// TIA Portal project "Plantilla_eProC" (V15.1)

(* hardware
DEVICE "S7-1200 station_1"  S7-1200 Station
   slot 0: "Rack_0"  S7-1200 Rack  Rack  V1.0
   slot 1: "PLC_1"  CPU 1214C DC/DC/DC  6ES7 214-1AG40-0XB0  V4.3
*)

// ===== PLC "PLC_1"  CPU 1214C DC/DC/DC =====

VAR_GLOBAL   // PLC tag table "Tabla de variables estándar"
   "System_Byte" AT %MB1 : Byte;
   "FirstScan" AT %M1.0 : Bool;
   "DiagStatusUpdate" AT %M1.1 : Bool;
   "AlwaysTRUE" AT %M1.2 : Bool;
   "AlwaysFALSE" AT %M1.3 : Bool;
   "Clock_Byte" AT %MB0 : Byte;
   "Clock_10Hz" AT %M0.0 : Bool;
   "Clock_5Hz" AT %M0.1 : Bool;
   "Clock_2.5Hz" AT %M0.2 : Bool;
   "Clock_2Hz" AT %M0.3 : Bool;
   "Clock_1.25Hz" AT %M0.4 : Bool;
   "Clock_1Hz" AT %M0.5 : Bool;
   "Clock_0.625Hz" AT %M0.6 : Bool;
   "Clock_0.5Hz" AT %M0.7 : Bool;
   "Marca_Manual" AT %M2.0 : Bool;
   "Marca_Automatico" AT %M2.1 : Bool;
   "Tim_Extrac_Rdy" AT %M3.0 : Bool;
   "Tim_Induc_Rdy" AT %M3.1 : Bool;
   "B_TimAperturaLados" AT %M4.0 : Bool;
END_VAR

VAR_GLOBAL   // PLC tag table "Entradas_PLC"
   "iPul_ParEmergencia" AT %I0.0 : Bool;
   "iSel_CicloManual" AT %I0.1 : Bool;
   "iSel_CicloAuto" AT %I0.2 : Bool;
   "iSel_AvanzCamaRolos1" AT %I0.3 : Bool;
   "iSel_RetroCamaRolos1" AT %I0.4 : Bool;
   "iSel_AvanzCamaRolos2" AT %I0.5 : Bool;
   "iSel_RetroCamaRolos2" AT %I0.6 : Bool;
   "iReserva1" AT %I0.7 : Bool;
   "iProt_TermicaRolos" AT %I1.0 : Bool;
   "iStart_CicloDesdeSoldad" AT %I1.1 : Bool;
   "iSns_PresAire" AT %I1.2 : Bool;
   "iReserva2" AT %I1.3 : Bool;
   "iReserva3" AT %I1.4 : Bool;
   "iReserva4" AT %I1.5 : Bool;
   "iSns_ElevArriba" AT %I2.0 : Bool;
   "iSns_ElevAbajo" AT %I2.1 : Bool;
   "iSns_ElevNormal" AT %I2.2 : Bool;
   "iSns_ElevRotado" AT %I2.3 : Bool;
   "iSns_PreseProduc" AT %I2.4 : Bool;
   "iSns_CR1LadoTableroArri" AT %I2.5 : Bool;
   "iSns_CR1LadoTableroAbaj" AT %I2.6 : Bool;
   "iSns_RegAlturaPaq" AT %I2.7 : Bool;
   "iSns_CR1LadoOpuesArri" AT %I3.0 : Bool;
   "iSns_CR1LadoOpuesAbaj" AT %I3.1 : Bool;
   "iSns_PreseProducSalida1" AT %I3.2 : Bool;
   "iSns_PreseProducSalida2" AT %I3.3 : Bool;
   "iPul_StartCiclo" AT %I3.4 : Bool;
   "iSel_HabRuedExtrac" AT %I3.5 : Bool;
   "iPul_MarchRuedExtrac" AT %I3.6 : Bool;
   "iReserva5" AT %I3.7 : Bool;
   "iSel_HabRuedIntroduc" AT %I4.0 : Bool;
   "iPul_MarchRuedIntroduc" AT %I4.1 : Bool;
END_VAR

VAR_GLOBAL   // PLC tag table "Salidas_PLC"
   "qCR1_LTArri" AT %Q0.0 : Bool;
   "qCR1_LTAbaj" AT %Q0.1 : Bool;
   "qCR1_LOArri" AT %Q0.2 : Bool;
   "qCR1_LOAbaj" AT %Q0.3 : Bool;
   "qCR1_Avance" AT %Q0.4 : Bool;
   "qCR1_Retroceso" AT %Q0.5 : Bool;
   "qCR2_Avance" AT %Q0.6 : Bool;
   "qCR2_Retroceso" AT %Q0.7 : Bool;
   "qHab_Comandos" AT %Q1.0 : Bool;
   "qRdy_VoltRdyaSold" AT %Q1.1 : Bool;
   "qBrk_Volt" AT %Q2.0 : Bool;
   "qBrk_Elev" AT %Q2.1 : Bool;
   "qCls_RodExtrac" AT %Q2.2 : Bool;
   "qCls_RodInduc" AT %Q2.3 : Bool;
   "qCls_Ganchos" AT %Q2.4 : Bool;
   "qOpn_Lados" AT %Q2.5 : Bool;
   "qAcc_Compact" AT %Q2.6 : Bool;
   "qCls_SoportRed" AT %Q2.7 : Bool;
END_VAR

DATA_BLOCK "DB_SUB_0_GENERAL"   // DB100
{ S7_Optimized_Access := 'TRUE' }
VERSION : 0.1
// stored: InstanceOfName FB_SUB_0_GENERAL
"FB_SUB_0_GENERAL"
BEGIN
END_DATA_BLOCK

DATA_BLOCK "DB_SUB_1_ELEVADOR"   // DB101
{ S7_Optimized_Access := 'TRUE' }
VERSION : 0.1
// stored: InstanceOfName FB_SUB_1_ELEVADOR
"FB_SUB_1_ELEVADOR"
BEGIN
END_DATA_BLOCK

DATA_BLOCK "DB_SUB_1_CAMAS_ROLOS"   // DB102
{ S7_Optimized_Access := 'TRUE' }
VERSION : 0.1
// stored: InstanceOfName FB_SUB_1_CAMAS_ROLOS
"FB_SUB_1_CAMAS_ROLOS"
BEGIN
END_DATA_BLOCK

DATA_BLOCK "DB_SUB_1_MAQUINA_ESTADOS_3"   // DB103
{ S7_Optimized_Access := 'TRUE' }
VERSION : 0.1
// stored: InstanceOfName FB_SUB_1_MAQUINA_ESTADOS_3
"FB_SUB_1_MAQUINA_ESTADOS_3"
BEGIN
END_DATA_BLOCK

DATA_BLOCK "DB_SUB_1_MAQUINA_ESTADOS_4"   // DB104
{ S7_Optimized_Access := 'TRUE' }
VERSION : 0.1
// stored: InstanceOfName FB_SUB_1_MAQUINA_ESTADOS_4
"FB_SUB_1_MAQUINA_ESTADOS_4"
BEGIN
END_DATA_BLOCK

// folder: AJUSTE_PEM

DATA_BLOCK "DB_SUB_0_PEM_GENERAL"   // DB400
{ S7_Optimized_Access := 'TRUE' }
VERSION : 0.1
BEGIN
END_DATA_BLOCK

DATA_BLOCK "DB_SUB_1_PEM_MAQ_ESTADO_1"   // DB401
{ S7_Optimized_Access := 'TRUE' }
VERSION : 0.1
BEGIN
END_DATA_BLOCK

DATA_BLOCK "DB_SUB_1_PEM_MAQ_ESTADO_2"   // DB402
{ S7_Optimized_Access := 'TRUE' }
VERSION : 0.1
BEGIN
END_DATA_BLOCK

DATA_BLOCK "DB_SUB_1_PEM_MAQ_ESTADO_3"   // DB403
{ S7_Optimized_Access := 'TRUE' }
VERSION : 0.1
BEGIN
END_DATA_BLOCK

DATA_BLOCK "DB_SUB_1_PEM_MAQ_ESTADO_4"   // DB404
{ S7_Optimized_Access := 'TRUE' }
VERSION : 0.1
BEGIN
END_DATA_BLOCK

// folder: COMANDOS

DATA_BLOCK "DB_SUB_0_COM_GENERAL"   // DB600
{ S7_Optimized_Access := 'TRUE' }
VERSION : 0.1
BEGIN
END_DATA_BLOCK

DATA_BLOCK "DB_SUB_1_COM_MAQ_ESTADO_1"   // DB601
{ S7_Optimized_Access := 'TRUE' }
VERSION : 0.1
BEGIN
END_DATA_BLOCK

DATA_BLOCK "DB_SUB_1_COM_MAQ_ESTADO_2"   // DB602
{ S7_Optimized_Access := 'TRUE' }
VERSION : 0.1
BEGIN
END_DATA_BLOCK

DATA_BLOCK "DB_SUB_1_COM_MAQ_ESTADO_3"   // DB603
{ S7_Optimized_Access := 'TRUE' }
VERSION : 0.1
BEGIN
END_DATA_BLOCK

DATA_BLOCK "DB_SUB_1_COM_MAQ_ESTADO_4"   // DB604
{ S7_Optimized_Access := 'TRUE' }
VERSION : 0.1
BEGIN
END_DATA_BLOCK

// folder: ENCLAVAMIENTOS

DATA_BLOCK "DB_SUB_0_ENC_GENERAL"   // DB700
{ S7_Optimized_Access := 'TRUE' }
VERSION : 0.1
BEGIN
END_DATA_BLOCK

DATA_BLOCK "DB_SUB_1_ENC_MAQ_ESTADOS_1"   // DB701
{ S7_Optimized_Access := 'TRUE' }
VERSION : 0.1
BEGIN
END_DATA_BLOCK

DATA_BLOCK "DB_SUB_1_ENC_MAQ_ESTADOS_2"   // DB702
{ S7_Optimized_Access := 'TRUE' }
VERSION : 0.1
BEGIN
END_DATA_BLOCK

DATA_BLOCK "DB_SUB_1_ENC_MAQ_ESTADOS_3"   // DB703
{ S7_Optimized_Access := 'TRUE' }
VERSION : 0.1
BEGIN
END_DATA_BLOCK

DATA_BLOCK "DB_SUB_1_ENC_MAQ_ESTADOS_4"   // DB704
{ S7_Optimized_Access := 'TRUE' }
VERSION : 0.1
BEGIN
END_DATA_BLOCK

// folder: ESTANDAR

DATA_BLOCK "Datos PLC"   // DB4
{ S7_Optimized_Access := 'TRUE' }
VERSION : 0.1
   VAR
      FH_Setpoint : DTL;   // Fecha y Hora del PLC
      FH : DTL;   // Fecha y Hora del PLC
      COM_Ajuste_FH : Bool;
   END_VAR
BEGIN
END_DATA_BLOCK

// folder: INCIDENTES

DATA_BLOCK "DB_SUB_0_GENERAL_ALARM"   // DB1100
{ S7_Optimized_Access := 'TRUE' }
VERSION : 0.1
// stored: InstanceOfName FB_SUB_0_GENERAL_ALARM
"FB_SUB_0_GENERAL_ALARM"
BEGIN
END_DATA_BLOCK

DATA_BLOCK "DB_SUB_1_MAQ_ESTADO_1_ALARM"   // DB1101
{ S7_Optimized_Access := 'TRUE' }
VERSION : 0.1
// stored: InstanceOfName FB_SUB_1_MAQ_ESTADO_1_ALARM
"FB_SUB_1_MAQ_ESTADO_1_ALARM"
BEGIN
END_DATA_BLOCK

DATA_BLOCK "DB_SUB_1_MAQ_ESTADO_2_ALARM"   // DB1102
{ S7_Optimized_Access := 'TRUE' }
VERSION : 0.1
// stored: InstanceOfName FB_SUB_1_MAQ_ESTADO_2_ALARM
"FB_SUB_1_MAQ_ESTADO_2_ALARM"
BEGIN
END_DATA_BLOCK

DATA_BLOCK "DB_SUB_1_MAQ_ESTADO_3_ALARM"   // DB1103
{ S7_Optimized_Access := 'TRUE' }
VERSION : 0.1
// stored: InstanceOfName FB_SUB_1_MAQ_ESTADO_3_ALARM
"FB_SUB_1_MAQ_ESTADO_3_ALARM"
BEGIN
END_DATA_BLOCK

DATA_BLOCK "DB_SUB_1_MAQ_ESTADO_4_ALARM"   // DB1104
{ S7_Optimized_Access := 'TRUE' }
VERSION : 0.1
// stored: InstanceOfName FB_SUB_1_MAQ_ESTADO_4_ALARM
"FB_SUB_1_MAQ_ESTADO_4_ALARM"
BEGIN
END_DATA_BLOCK

// folder: MECANICA

DATA_BLOCK "DB_SUB_0_MEC_GENERAL"   // DB300
{ S7_Optimized_Access := 'TRUE' }
VERSION : 0.1
BEGIN
END_DATA_BLOCK

DATA_BLOCK "DB_SUB_1_MEC_MAQ_ESTADO_1"   // DB301
{ S7_Optimized_Access := 'TRUE' }
VERSION : 0.1
BEGIN
END_DATA_BLOCK

DATA_BLOCK "DB_SUB_1_MEC_MAQ_ESTADO_2"   // DB302
{ S7_Optimized_Access := 'TRUE' }
VERSION : 0.1
BEGIN
END_DATA_BLOCK

DATA_BLOCK "DB_SUB_1_MEC_MAQ_ESTADO_3"   // DB303
{ S7_Optimized_Access := 'TRUE' }
VERSION : 0.1
BEGIN
END_DATA_BLOCK

DATA_BLOCK "DB_SUB_1_MEC_MAQ_ESTADO_4"   // DB304
{ S7_Optimized_Access := 'TRUE' }
VERSION : 0.1
BEGIN
END_DATA_BLOCK

// folder: System blocks/Program resources

DATA_BLOCK "IEC_Timer_0_DB"   // DB1
{ S7_Optimized_Access := 'TRUE' }
AUTHOR : Simatic
FAMILY : IEC
NAME : IEC_TMR
VERSION : 1.0
// stored: InstanceOfName IEC_TIMER
"IEC_TIMER"
BEGIN
END_DATA_BLOCK

DATA_BLOCK "IEC_Timer_1_DB"   // DB2
{ S7_Optimized_Access := 'TRUE' }
AUTHOR : Simatic
FAMILY : IEC
NAME : IEC_TMR
VERSION : 1.0
// stored: InstanceOfName IEC_TIMER
"IEC_TIMER"
BEGIN
END_DATA_BLOCK

DATA_BLOCK "IEC_Timer_2_DB"   // DB3
{ S7_Optimized_Access := 'TRUE' }
AUTHOR : Simatic
FAMILY : IEC
NAME : IEC_TMR
VERSION : 1.0
// stored: InstanceOfName IEC_TIMER
"IEC_TIMER"
BEGIN
END_DATA_BLOCK

DATA_BLOCK "IEC_Timer_3_DB"   // DB5
{ S7_Optimized_Access := 'TRUE' }
AUTHOR : Simatic
FAMILY : IEC
NAME : IEC_TMR
VERSION : 1.0
// stored: InstanceOfName IEC_TIMER
"IEC_TIMER"
BEGIN
END_DATA_BLOCK

DATA_BLOCK "IEC_Timer_5_DB"   // DB6
{ S7_Optimized_Access := 'TRUE' }
AUTHOR : Simatic
FAMILY : IEC
NAME : IEC_TMR
VERSION : 1.0
// stored: InstanceOfName IEC_TIMER
"IEC_TIMER"
BEGIN
END_DATA_BLOCK

DATA_BLOCK "IEC_Timer_6_DB"   // DB7
{ S7_Optimized_Access := 'TRUE' }
AUTHOR : Simatic
FAMILY : IEC
NAME : IEC_TMR
VERSION : 1.0
// stored: InstanceOfName IEC_TIMER
"IEC_TIMER"
BEGIN
END_DATA_BLOCK

DATA_BLOCK "IEC_Timer_7_DB"   // DB8
{ S7_Optimized_Access := 'TRUE' }
AUTHOR : Simatic
FAMILY : IEC
NAME : IEC_TMR
VERSION : 1.0
// stored: InstanceOfName IEC_TIMER
"IEC_TIMER"
BEGIN
END_DATA_BLOCK

// folder: VISUALIZACION

DATA_BLOCK "DB_SUB_0_VIS_GENERAL"   // DB800
{ S7_Optimized_Access := 'TRUE' }
VERSION : 0.1
BEGIN
END_DATA_BLOCK

DATA_BLOCK "DB_SUB_1_VIS_MAQ_ESTADO_1"   // DB801
{ S7_Optimized_Access := 'TRUE' }
VERSION : 0.1
BEGIN
END_DATA_BLOCK

DATA_BLOCK "DB_SUB_1_VIS_MAQ_ESTADO_2"   // DB802
{ S7_Optimized_Access := 'TRUE' }
VERSION : 0.1
BEGIN
END_DATA_BLOCK

DATA_BLOCK "DB_SUB_1_VIS_MAQ_ESTADO_3"   // DB803
{ S7_Optimized_Access := 'TRUE' }
VERSION : 0.1
BEGIN
END_DATA_BLOCK

DATA_BLOCK "DB_SUB_1_VIS_MAQ_ESTADO_4"   // DB804
{ S7_Optimized_Access := 'TRUE' }
VERSION : 0.1
BEGIN
END_DATA_BLOCK

// folder: (top level)

FUNCTION_BLOCK "FB_SUB_0_GENERAL"   // FB100, LAD
{ S7_Optimized_Access := 'TRUE' }
VERSION : 0.1
BEGIN

REGION Network 1: Instanciado Bloque "FB_SUB_1_MAQUINA_ESTADOS_1"
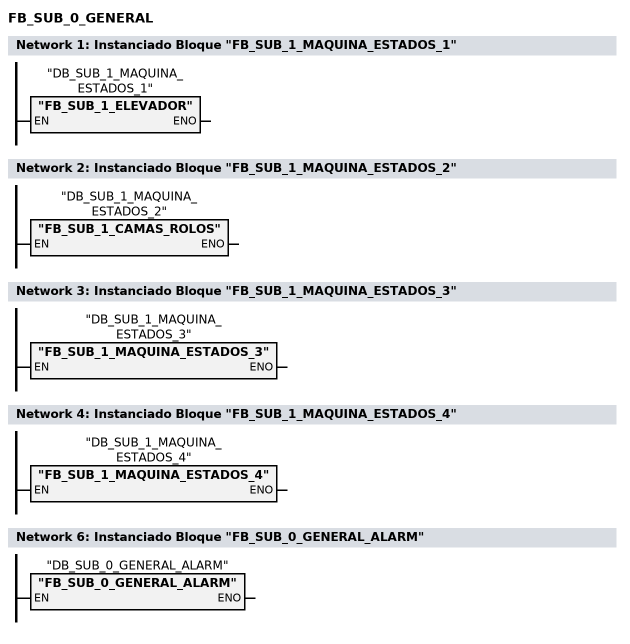
   RUNG wire#powerrail
      "DB_SUB_1_MAQUINA_ESTADOS_1"()
   END_RUNG
   // the same network as SCL:
   "DB_SUB_1_MAQUINA_ESTADOS_1"();   // "FB_SUB_1_ELEVADOR"
END_REGION

REGION Network 2: Instanciado Bloque "FB_SUB_1_MAQUINA_ESTADOS_2"
   RUNG wire#powerrail
      "DB_SUB_1_MAQUINA_ESTADOS_2"()
   END_RUNG
   // the same network as SCL:
   "DB_SUB_1_MAQUINA_ESTADOS_2"();   // "FB_SUB_1_CAMAS_ROLOS"
END_REGION

REGION Network 3: Instanciado Bloque "FB_SUB_1_MAQUINA_ESTADOS_3"
   RUNG wire#powerrail
      "DB_SUB_1_MAQUINA_ESTADOS_3"()
   END_RUNG
   // the same network as SCL:
   "DB_SUB_1_MAQUINA_ESTADOS_3"();   // "FB_SUB_1_MAQUINA_ESTADOS_3"
END_REGION

REGION Network 4: Instanciado Bloque "FB_SUB_1_MAQUINA_ESTADOS_4"
   RUNG wire#powerrail
      "DB_SUB_1_MAQUINA_ESTADOS_4"()
   END_RUNG
   // the same network as SCL:
   "DB_SUB_1_MAQUINA_ESTADOS_4"();   // "FB_SUB_1_MAQUINA_ESTADOS_4"
END_REGION

REGION Network 5: ---------------------------------------------------------------------------------------------------------
END_REGION

REGION Network 6: Instanciado Bloque "FB_SUB_0_GENERAL_ALARM"
   RUNG wire#powerrail
      "DB_SUB_0_GENERAL_ALARM"()
   END_RUNG
   // the same network as SCL:
   "DB_SUB_0_GENERAL_ALARM"();   // "FB_SUB_0_GENERAL_ALARM"
END_REGION
END_FUNCTION_BLOCK

FUNCTION_BLOCK "FB_SUB_1_ELEVADOR"   // FB101, LAD
{ S7_Optimized_Access := 'TRUE' }
VERSION : 0.1
   VAR
      Estados : Array[0..32] of Bool;
      Concatenadoras : Array[0..32] of Bool;
      Prioritarias : Array[0..32] of Bool;
   END_VAR
BEGIN

REGION Network 1: --------------------------------------INSTANCIADO DE SUBSISTEMAS ---------------------------------------------------------
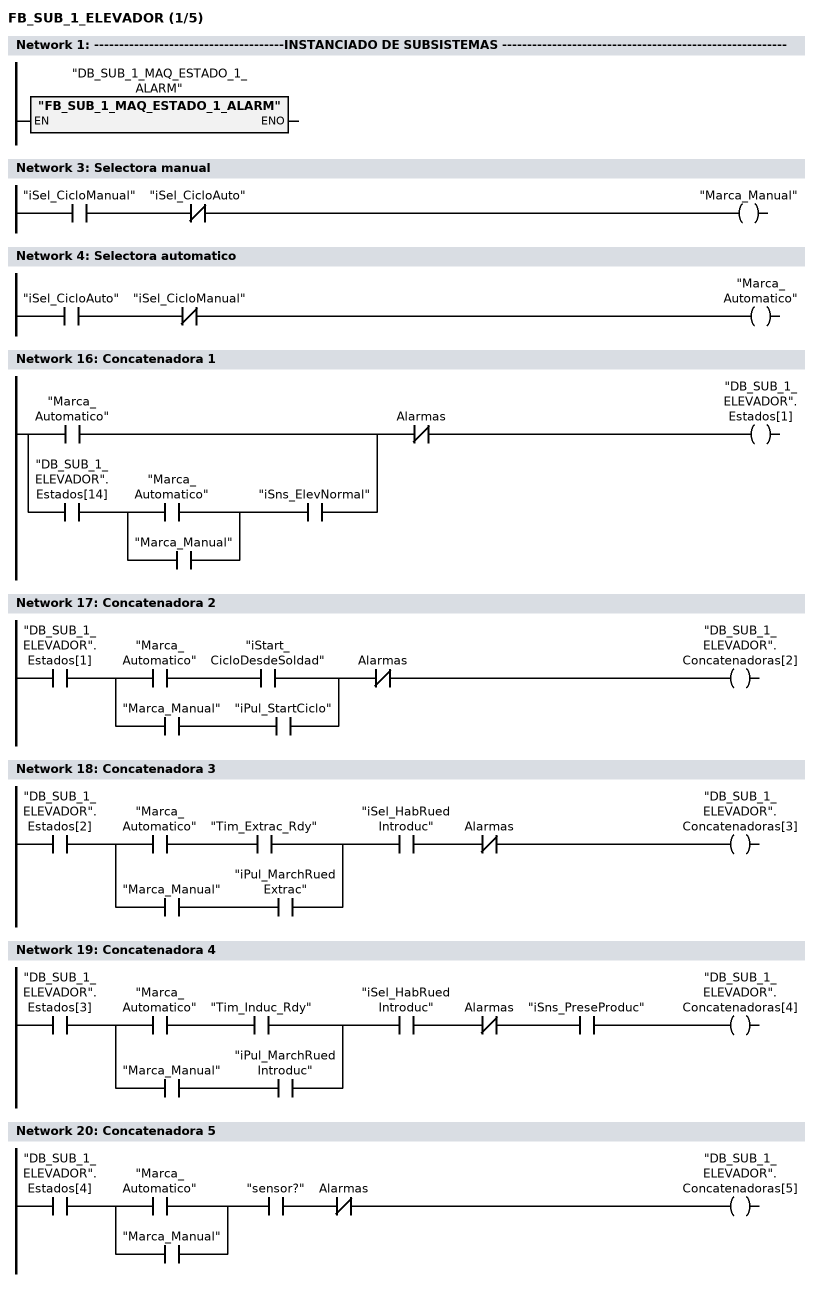
   RUNG wire#powerrail
      "DB_SUB_1_MAQ_ESTADO_1_ALARM"()
   END_RUNG
   // the same network as SCL:
   "DB_SUB_1_MAQ_ESTADO_1_ALARM"();   // "FB_SUB_1_MAQ_ESTADO_1_ALARM"
END_REGION

REGION Network 2: ------------------------------ ESTADOS DE LA MAQUINA - auto/manual -------------------------------------
END_REGION

REGION Network 3: Selectora manual
   RUNG wire#powerrail
      Contact( "iSel_CicloManual" )
      I_Contact( "iSel_CicloAuto" )
      Coil( "Marca_Manual" )
   END_RUNG
   // the same network as SCL:
   "Marca_Manual" := "iSel_CicloManual" AND NOT "iSel_CicloAuto";
END_REGION

REGION Network 4: Selectora automatico
   RUNG wire#powerrail
      Contact( "iSel_CicloAuto" )
      I_Contact( "iSel_CicloManual" )
      Coil( "Marca_Automatico" )
   END_RUNG
   // the same network as SCL:
   "Marca_Automatico" := "iSel_CicloAuto" AND NOT "iSel_CicloManual";
END_REGION

REGION Network 8: --------------------------------------OTROS ---------------------------------------------------------
END_REGION

REGION Network 15: --------------------------------------MAQUINA DE ESTADOS ---------------------------------------------------------
END_REGION

REGION Network 16: Concatenadora 1
   RUNG wire#powerrail
      Contact( "Marca_Automatico" )
      wire#w1
      I_Contact( Alarmas )
      Coil( "DB_SUB_1_ELEVADOR".Estados[1] )
   END_RUNG
   RUNG wire#powerrail
      Contact( "DB_SUB_1_ELEVADOR".Estados[14] )
      wire#w2
      Contact( "Marca_Automatico" )
      wire#w3
      Contact( "iSns_ElevNormal" )
   END_RUNG wire#w1
   RUNG wire#w2
      Contact( "Marca_Manual" )
   END_RUNG wire#w3
   // the same network as SCL:
   "DB_SUB_1_ELEVADOR".Estados[1] := ("Marca_Automatico" OR ("DB_SUB_1_ELEVADOR".Estados[14] AND ("Marca_Automatico" OR "Marca_Manual") AND "iSns_ElevNormal")) AND NOT Alarmas;
END_REGION

REGION Network 17: Concatenadora 2
   RUNG wire#powerrail
      Contact( "DB_SUB_1_ELEVADOR".Estados[1] )
      wire#w1
      Contact( "Marca_Automatico" )
      Contact( "iStart_CicloDesdeSoldad" )
      wire#w2
      I_Contact( Alarmas )
      Coil( "DB_SUB_1_ELEVADOR".Concatenadoras[2] )
   END_RUNG
   RUNG wire#w1
      Contact( "Marca_Manual" )
      Contact( "iPul_StartCiclo" )
   END_RUNG wire#w2
   // the same network as SCL:
   "DB_SUB_1_ELEVADOR".Concatenadoras[2] := "DB_SUB_1_ELEVADOR".Estados[1] AND (("Marca_Automatico" AND "iStart_CicloDesdeSoldad") OR ("Marca_Manual" AND "iPul_StartCiclo")) AND NOT Alarmas;
END_REGION

REGION Network 18: Concatenadora 3
   RUNG wire#powerrail
      Contact( "DB_SUB_1_ELEVADOR".Estados[2] )
      wire#w1
      Contact( "Marca_Automatico" )
      Contact( "Tim_Extrac_Rdy" )
      wire#w2
      Contact( "iSel_HabRuedIntroduc" )
      I_Contact( Alarmas )
      Coil( "DB_SUB_1_ELEVADOR".Concatenadoras[3] )
   END_RUNG
   RUNG wire#w1
      Contact( "Marca_Manual" )
      Contact( "iPul_MarchRuedExtrac" )
   END_RUNG wire#w2
   // the same network as SCL:
   "DB_SUB_1_ELEVADOR".Concatenadoras[3] := "DB_SUB_1_ELEVADOR".Estados[2] AND (("Marca_Automatico" AND "Tim_Extrac_Rdy") OR ("Marca_Manual" AND "iPul_MarchRuedExtrac")) AND "iSel_HabRuedIntroduc" AND NOT Alarmas;
END_REGION

REGION Network 19: Concatenadora 4
   RUNG wire#powerrail
      Contact( "DB_SUB_1_ELEVADOR".Estados[3] )
      wire#w1
      Contact( "Marca_Automatico" )
      Contact( "Tim_Induc_Rdy" )
      wire#w2
      Contact( "iSel_HabRuedIntroduc" )
      I_Contact( Alarmas )
      Contact( "iSns_PreseProduc" )
      Coil( "DB_SUB_1_ELEVADOR".Concatenadoras[4] )
   END_RUNG
   RUNG wire#w1
      Contact( "Marca_Manual" )
      Contact( "iPul_MarchRuedIntroduc" )
   END_RUNG wire#w2
   // the same network as SCL:
   "DB_SUB_1_ELEVADOR".Concatenadoras[4] := "DB_SUB_1_ELEVADOR".Estados[3] AND (("Marca_Automatico" AND "Tim_Induc_Rdy") OR ("Marca_Manual" AND "iPul_MarchRuedIntroduc")) AND "iSel_HabRuedIntroduc" AND NOT Alarmas AND "iSns_PreseProduc";
END_REGION

REGION Network 20: Concatenadora 5
   RUNG wire#powerrail
      Contact( "DB_SUB_1_ELEVADOR".Estados[4] )
      wire#w1
      Contact( "Marca_Automatico" )
      wire#w2
      Contact( "sensor?" )
      I_Contact( Alarmas )
      Coil( "DB_SUB_1_ELEVADOR".Concatenadoras[5] )
   END_RUNG
   RUNG wire#w1
      Contact( "Marca_Manual" )
   END_RUNG wire#w2
   // the same network as SCL:
   "DB_SUB_1_ELEVADOR".Concatenadoras[5] := "DB_SUB_1_ELEVADOR".Estados[4] AND ("Marca_Automatico" OR "Marca_Manual") AND "sensor?" AND NOT Alarmas;
END_REGION

REGION Network 21: Concatenadora 6
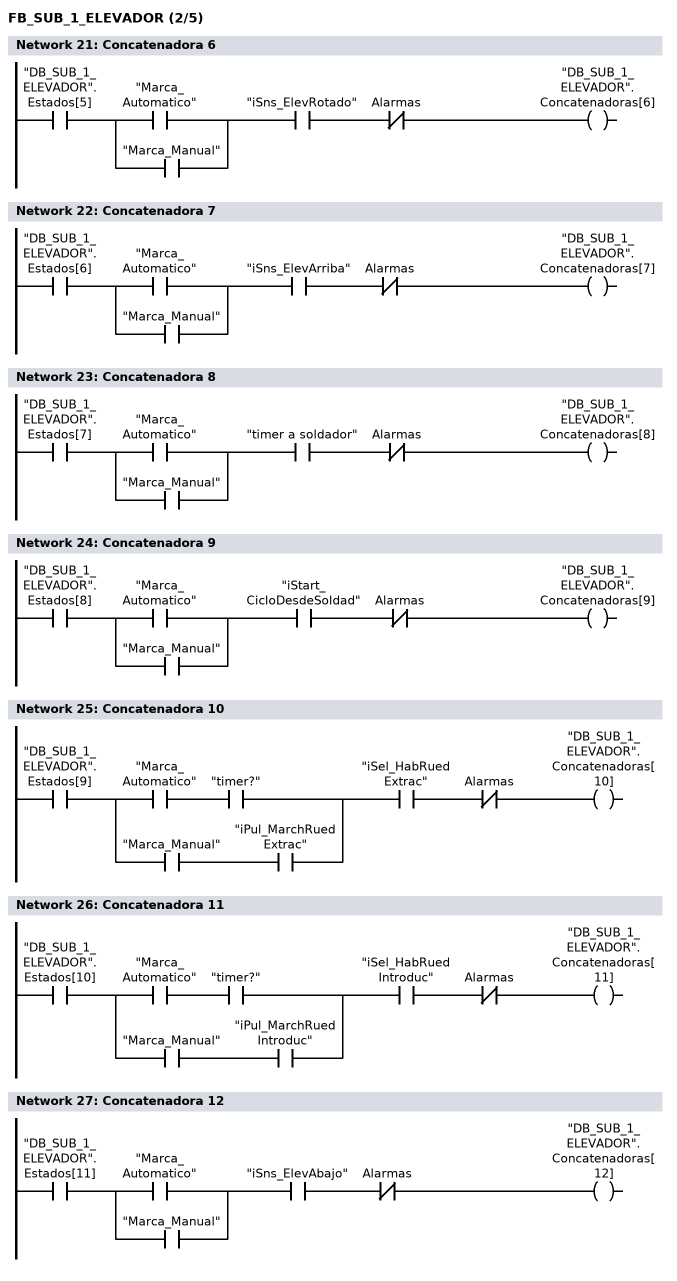
   RUNG wire#powerrail
      Contact( "DB_SUB_1_ELEVADOR".Estados[5] )
      wire#w1
      Contact( "Marca_Automatico" )
      wire#w2
      Contact( "iSns_ElevRotado" )
      I_Contact( Alarmas )
      Coil( "DB_SUB_1_ELEVADOR".Concatenadoras[6] )
   END_RUNG
   RUNG wire#w1
      Contact( "Marca_Manual" )
   END_RUNG wire#w2
   // the same network as SCL:
   "DB_SUB_1_ELEVADOR".Concatenadoras[6] := "DB_SUB_1_ELEVADOR".Estados[5] AND ("Marca_Automatico" OR "Marca_Manual") AND "iSns_ElevRotado" AND NOT Alarmas;
END_REGION

REGION Network 22: Concatenadora 7
   RUNG wire#powerrail
      Contact( "DB_SUB_1_ELEVADOR".Estados[6] )
      wire#w1
      Contact( "Marca_Automatico" )
      wire#w2
      Contact( "iSns_ElevArriba" )
      I_Contact( Alarmas )
      Coil( "DB_SUB_1_ELEVADOR".Concatenadoras[7] )
   END_RUNG
   RUNG wire#w1
      Contact( "Marca_Manual" )
   END_RUNG wire#w2
   // the same network as SCL:
   "DB_SUB_1_ELEVADOR".Concatenadoras[7] := "DB_SUB_1_ELEVADOR".Estados[6] AND ("Marca_Automatico" OR "Marca_Manual") AND "iSns_ElevArriba" AND NOT Alarmas;
END_REGION

REGION Network 23: Concatenadora 8
   RUNG wire#powerrail
      Contact( "DB_SUB_1_ELEVADOR".Estados[7] )
      wire#w1
      Contact( "Marca_Automatico" )
      wire#w2
      Contact( "timer a soldador" )
      I_Contact( Alarmas )
      Coil( "DB_SUB_1_ELEVADOR".Concatenadoras[8] )
   END_RUNG
   RUNG wire#w1
      Contact( "Marca_Manual" )
   END_RUNG wire#w2
   // the same network as SCL:
   "DB_SUB_1_ELEVADOR".Concatenadoras[8] := "DB_SUB_1_ELEVADOR".Estados[7] AND ("Marca_Automatico" OR "Marca_Manual") AND "timer a soldador" AND NOT Alarmas;
END_REGION

REGION Network 24: Concatenadora 9
   RUNG wire#powerrail
      Contact( "DB_SUB_1_ELEVADOR".Estados[8] )
      wire#w1
      Contact( "Marca_Automatico" )
      wire#w2
      Contact( "iStart_CicloDesdeSoldad" )
      I_Contact( Alarmas )
      Coil( "DB_SUB_1_ELEVADOR".Concatenadoras[9] )
   END_RUNG
   RUNG wire#w1
      Contact( "Marca_Manual" )
   END_RUNG wire#w2
   // the same network as SCL:
   "DB_SUB_1_ELEVADOR".Concatenadoras[9] := "DB_SUB_1_ELEVADOR".Estados[8] AND ("Marca_Automatico" OR "Marca_Manual") AND "iStart_CicloDesdeSoldad" AND NOT Alarmas;
END_REGION

REGION Network 25: Concatenadora 10
   RUNG wire#powerrail
      Contact( "DB_SUB_1_ELEVADOR".Estados[9] )
      wire#w1
      Contact( "Marca_Automatico" )
      Contact( "timer?" )
      wire#w2
      Contact( "iSel_HabRuedExtrac" )
      I_Contact( Alarmas )
      Coil( "DB_SUB_1_ELEVADOR".Concatenadoras[10] )
   END_RUNG
   RUNG wire#w1
      Contact( "Marca_Manual" )
      Contact( "iPul_MarchRuedExtrac" )
   END_RUNG wire#w2
   // the same network as SCL:
   "DB_SUB_1_ELEVADOR".Concatenadoras[10] := "DB_SUB_1_ELEVADOR".Estados[9] AND (("Marca_Automatico" AND "timer?") OR ("Marca_Manual" AND "iPul_MarchRuedExtrac")) AND "iSel_HabRuedExtrac" AND NOT Alarmas;
END_REGION

REGION Network 26: Concatenadora 11
   RUNG wire#powerrail
      Contact( "DB_SUB_1_ELEVADOR".Estados[10] )
      wire#w1
      Contact( "Marca_Automatico" )
      Contact( "timer?" )
      wire#w2
      Contact( "iSel_HabRuedIntroduc" )
      I_Contact( Alarmas )
      Coil( "DB_SUB_1_ELEVADOR".Concatenadoras[11] )
   END_RUNG
   RUNG wire#w1
      Contact( "Marca_Manual" )
      Contact( "iPul_MarchRuedIntroduc" )
   END_RUNG wire#w2
   // the same network as SCL:
   "DB_SUB_1_ELEVADOR".Concatenadoras[11] := "DB_SUB_1_ELEVADOR".Estados[10] AND (("Marca_Automatico" AND "timer?") OR ("Marca_Manual" AND "iPul_MarchRuedIntroduc")) AND "iSel_HabRuedIntroduc" AND NOT Alarmas;
END_REGION

REGION Network 27: Concatenadora 12
   RUNG wire#powerrail
      Contact( "DB_SUB_1_ELEVADOR".Estados[11] )
      wire#w1
      Contact( "Marca_Automatico" )
      wire#w2
      Contact( "iSns_ElevAbajo" )
      I_Contact( Alarmas )
      Coil( "DB_SUB_1_ELEVADOR".Concatenadoras[12] )
   END_RUNG
   RUNG wire#w1
      Contact( "Marca_Manual" )
   END_RUNG wire#w2
   // the same network as SCL:
   "DB_SUB_1_ELEVADOR".Concatenadoras[12] := "DB_SUB_1_ELEVADOR".Estados[11] AND ("Marca_Automatico" OR "Marca_Manual") AND "iSns_ElevAbajo" AND NOT Alarmas;
END_REGION

REGION Network 28: Concatenadora 13
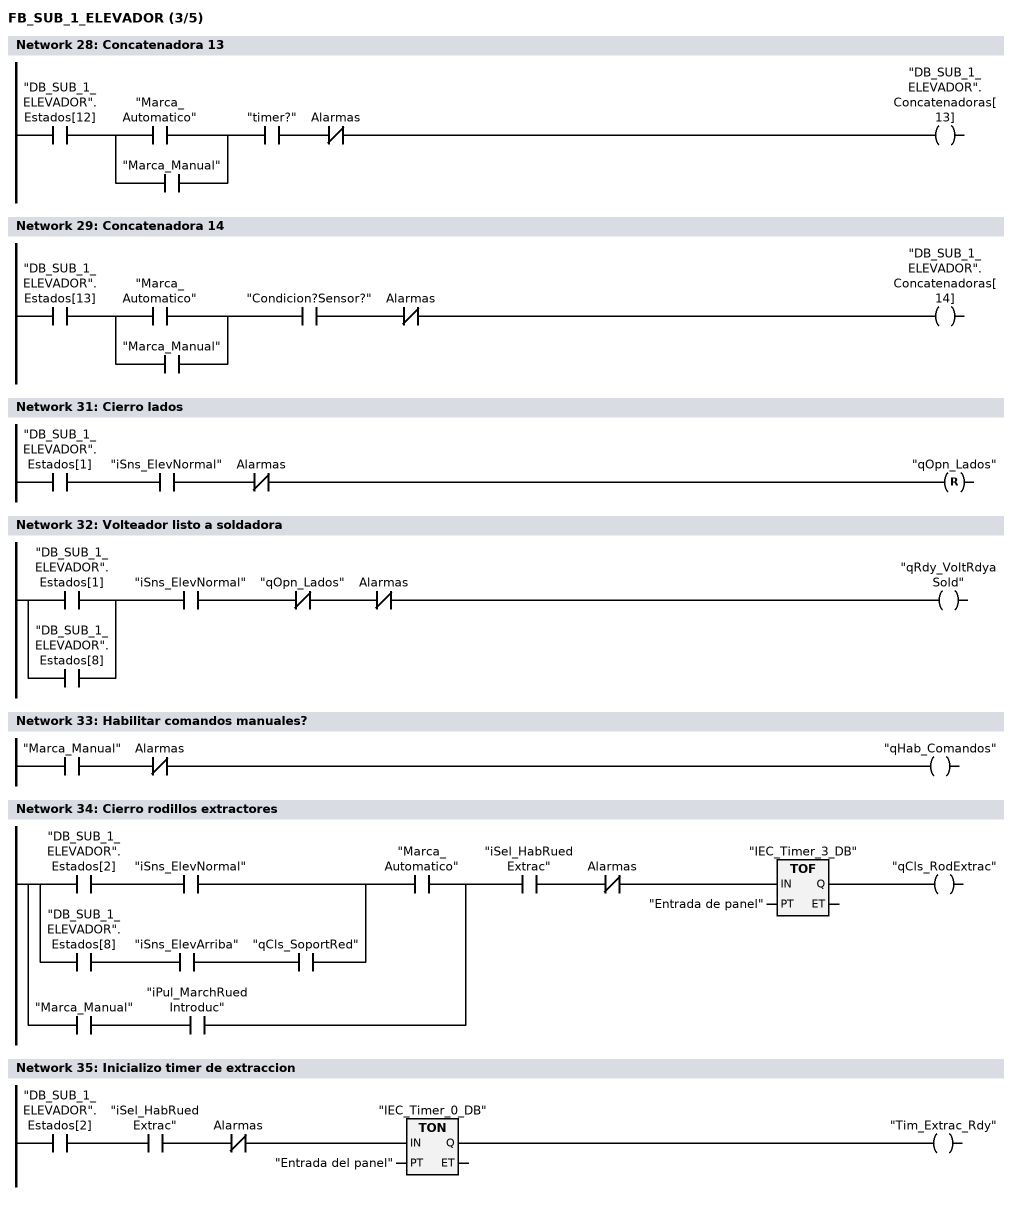
   RUNG wire#powerrail
      Contact( "DB_SUB_1_ELEVADOR".Estados[12] )
      wire#w1
      Contact( "Marca_Automatico" )
      wire#w2
      Contact( "timer?" )
      I_Contact( Alarmas )
      Coil( "DB_SUB_1_ELEVADOR".Concatenadoras[13] )
   END_RUNG
   RUNG wire#w1
      Contact( "Marca_Manual" )
   END_RUNG wire#w2
   // the same network as SCL:
   "DB_SUB_1_ELEVADOR".Concatenadoras[13] := "DB_SUB_1_ELEVADOR".Estados[12] AND ("Marca_Automatico" OR "Marca_Manual") AND "timer?" AND NOT Alarmas;
END_REGION

REGION Network 29: Concatenadora 14
   RUNG wire#powerrail
      Contact( "DB_SUB_1_ELEVADOR".Estados[13] )
      wire#w1
      Contact( "Marca_Automatico" )
      wire#w2
      Contact( "Condicion?Sensor?" )
      I_Contact( Alarmas )
      Coil( "DB_SUB_1_ELEVADOR".Concatenadoras[14] )
   END_RUNG
   RUNG wire#w1
      Contact( "Marca_Manual" )
   END_RUNG wire#w2
   // the same network as SCL:
   "DB_SUB_1_ELEVADOR".Concatenadoras[14] := "DB_SUB_1_ELEVADOR".Estados[13] AND ("Marca_Automatico" OR "Marca_Manual") AND "Condicion?Sensor?" AND NOT Alarmas;
END_REGION

REGION Network 30: --------------------------------------ACCIONAMIENTOS ---------------------------------------------------------
END_REGION

REGION Network 31: Cierro lados
   RUNG wire#powerrail
      Contact( "DB_SUB_1_ELEVADOR".Estados[1] )
      Contact( "iSns_ElevNormal" )
      I_Contact( Alarmas )
      R_Coil( "qOpn_Lados" )
   END_RUNG
   // the same network as SCL:
   IF "DB_SUB_1_ELEVADOR".Estados[1] AND "iSns_ElevNormal" AND NOT Alarmas THEN
       "qOpn_Lados" := FALSE;
   END_IF;
END_REGION

REGION Network 32: Volteador listo a soldadora
   RUNG wire#powerrail
      Contact( "DB_SUB_1_ELEVADOR".Estados[1] )
      wire#w1
      Contact( "iSns_ElevNormal" )
      I_Contact( "qOpn_Lados" )
      I_Contact( Alarmas )
      Coil( "qRdy_VoltRdyaSold" )
   END_RUNG
   RUNG wire#powerrail
      Contact( "DB_SUB_1_ELEVADOR".Estados[8] )
   END_RUNG wire#w1
   // the same network as SCL:
   "qRdy_VoltRdyaSold" := ("DB_SUB_1_ELEVADOR".Estados[1] OR "DB_SUB_1_ELEVADOR".Estados[8]) AND "iSns_ElevNormal" AND NOT "qOpn_Lados" AND NOT Alarmas;
END_REGION

REGION Network 33: Habilitar comandos manuales?
   RUNG wire#powerrail
      Contact( "Marca_Manual" )
      I_Contact( Alarmas )
      Coil( "qHab_Comandos" )
   END_RUNG
   // the same network as SCL:
   "qHab_Comandos" := "Marca_Manual" AND NOT Alarmas;
END_REGION

REGION Network 34: Cierro rodillos extractores
   "IEC_Timer_3_DB".TOF(IN := (((("DB_SUB_1_ELEVADOR".Estados[2] AND "iSns_ElevNormal") OR ("DB_SUB_1_ELEVADOR".Estados[8] AND "iSns_ElevArriba" AND "qCls_SoportRed")) AND "Marca_Automatico") OR ("Marca_Manual" AND "iPul_MarchRuedIntroduc")) AND "iSel_HabRuedExtrac" AND NOT Alarmas,
                        PT := "Entrada de panel");
   "qCls_RodExtrac" := "IEC_Timer_3_DB".Q;
END_REGION

REGION Network 35: Inicializo timer de extraccion
   "IEC_Timer_0_DB".TON(IN := "DB_SUB_1_ELEVADOR".Estados[2] AND "iSel_HabRuedExtrac" AND NOT Alarmas,
                        PT := "Entrada del panel");
   "Tim_Extrac_Rdy" := "IEC_Timer_0_DB".Q;
END_REGION

REGION Network 36: Cierro rodillos inductores
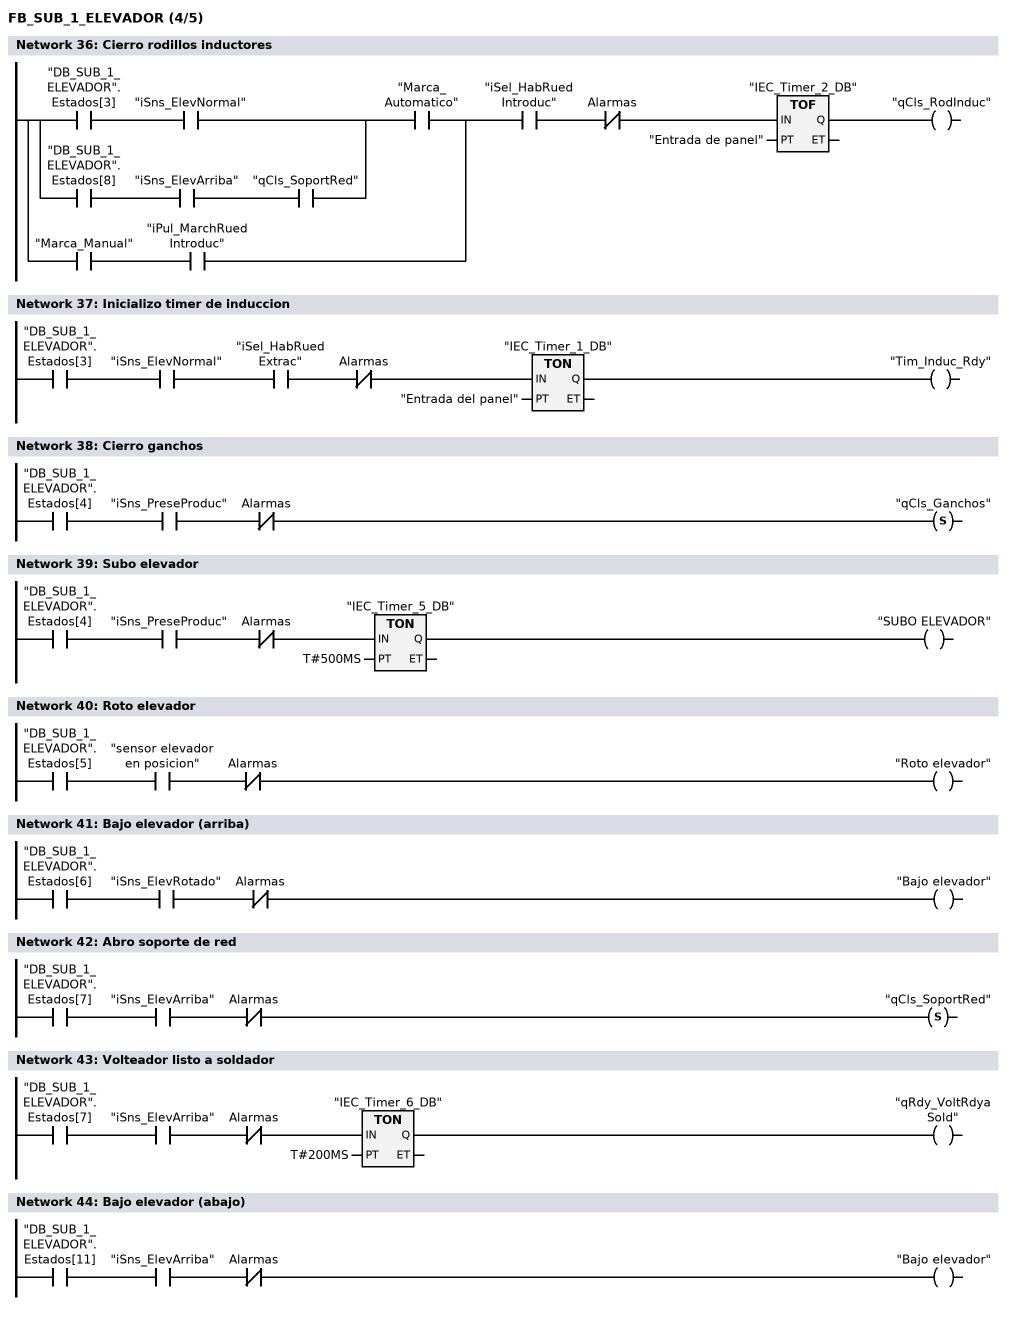
   "IEC_Timer_2_DB".TOF(IN := (((("DB_SUB_1_ELEVADOR".Estados[3] AND "iSns_ElevNormal") OR ("DB_SUB_1_ELEVADOR".Estados[8] AND "iSns_ElevArriba" AND "qCls_SoportRed")) AND "Marca_Automatico") OR ("Marca_Manual" AND "iPul_MarchRuedIntroduc")) AND "iSel_HabRuedIntroduc" AND NOT Alarmas,
                        PT := "Entrada de panel");
   "qCls_RodInduc" := "IEC_Timer_2_DB".Q;
END_REGION

REGION Network 37: Inicializo timer de induccion
   "IEC_Timer_1_DB".TON(IN := "DB_SUB_1_ELEVADOR".Estados[3] AND "iSns_ElevNormal" AND "iSel_HabRuedExtrac" AND NOT Alarmas,
                        PT := "Entrada del panel");
   "Tim_Induc_Rdy" := "IEC_Timer_1_DB".Q;
END_REGION

REGION Network 38: Cierro ganchos
   RUNG wire#powerrail
      Contact( "DB_SUB_1_ELEVADOR".Estados[4] )
      Contact( "iSns_PreseProduc" )
      I_Contact( Alarmas )
      S_Coil( "qCls_Ganchos" )
   END_RUNG
   // the same network as SCL:
   IF "DB_SUB_1_ELEVADOR".Estados[4] AND "iSns_PreseProduc" AND NOT Alarmas THEN
       "qCls_Ganchos" := TRUE;
   END_IF;
END_REGION

REGION Network 39: Subo elevador
   "IEC_Timer_5_DB".TON(IN := "DB_SUB_1_ELEVADOR".Estados[4] AND "iSns_PreseProduc" AND NOT Alarmas,
                        PT := T#500MS);
   "SUBO ELEVADOR" := "IEC_Timer_5_DB".Q;
END_REGION

REGION Network 40: Roto elevador
   RUNG wire#powerrail
      Contact( "DB_SUB_1_ELEVADOR".Estados[5] )
      Contact( "sensor elevador en posicion" )
      I_Contact( Alarmas )
      Coil( "Roto elevador" )
   END_RUNG
   // the same network as SCL:
   "Roto elevador" := "DB_SUB_1_ELEVADOR".Estados[5] AND "sensor elevador en posicion" AND NOT Alarmas;
END_REGION

REGION Network 41: Bajo elevador (arriba)
   RUNG wire#powerrail
      Contact( "DB_SUB_1_ELEVADOR".Estados[6] )
      Contact( "iSns_ElevRotado" )
      I_Contact( Alarmas )
      Coil( "Bajo elevador" )
   END_RUNG
   // the same network as SCL:
   "Bajo elevador" := "DB_SUB_1_ELEVADOR".Estados[6] AND "iSns_ElevRotado" AND NOT Alarmas;
END_REGION

REGION Network 42: Abro soporte de red
   RUNG wire#powerrail
      Contact( "DB_SUB_1_ELEVADOR".Estados[7] )
      Contact( "iSns_ElevArriba" )
      I_Contact( Alarmas )
      S_Coil( "qCls_SoportRed" )
   END_RUNG
   // the same network as SCL:
   IF "DB_SUB_1_ELEVADOR".Estados[7] AND "iSns_ElevArriba" AND NOT Alarmas THEN
       "qCls_SoportRed" := TRUE;
   END_IF;
END_REGION

REGION Network 43: Volteador listo a soldador
   "IEC_Timer_6_DB".TON(IN := "DB_SUB_1_ELEVADOR".Estados[7] AND "iSns_ElevArriba" AND NOT Alarmas,
                        PT := T#200MS);
   "qRdy_VoltRdyaSold" := "IEC_Timer_6_DB".Q;
END_REGION

REGION Network 44: Bajo elevador (abajo)
   RUNG wire#powerrail
      Contact( "DB_SUB_1_ELEVADOR".Estados[11] )
      Contact( "iSns_ElevArriba" )
      I_Contact( Alarmas )
      Coil( "Bajo elevador" )
   END_RUNG
   // the same network as SCL:
   "Bajo elevador" := "DB_SUB_1_ELEVADOR".Estados[11] AND "iSns_ElevArriba" AND NOT Alarmas;
END_REGION

REGION Network 45: Abro ganchos
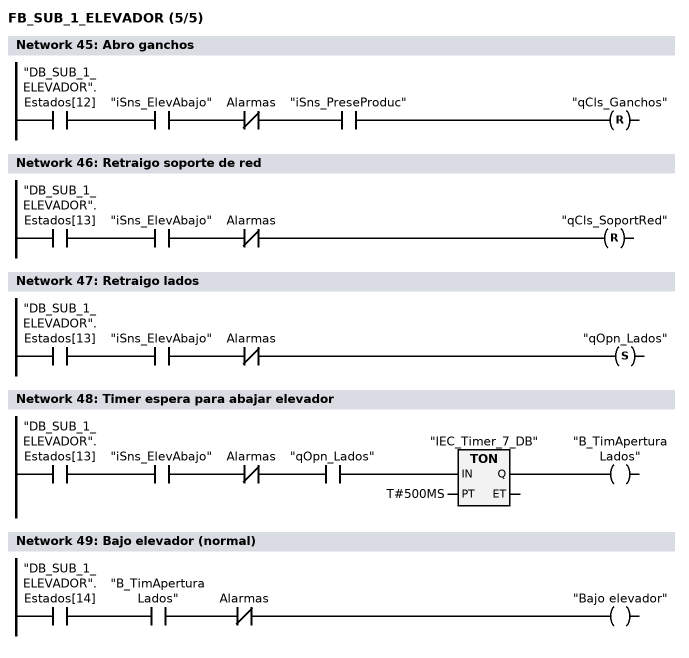
   RUNG wire#powerrail
      Contact( "DB_SUB_1_ELEVADOR".Estados[12] )
      Contact( "iSns_ElevAbajo" )
      I_Contact( Alarmas )
      Contact( "iSns_PreseProduc" )
      R_Coil( "qCls_Ganchos" )
   END_RUNG
   // the same network as SCL:
   IF "DB_SUB_1_ELEVADOR".Estados[12] AND "iSns_ElevAbajo" AND NOT Alarmas AND "iSns_PreseProduc" THEN
       "qCls_Ganchos" := FALSE;
   END_IF;
END_REGION

REGION Network 46: Retraigo soporte de red
   RUNG wire#powerrail
      Contact( "DB_SUB_1_ELEVADOR".Estados[13] )
      Contact( "iSns_ElevAbajo" )
      I_Contact( Alarmas )
      R_Coil( "qCls_SoportRed" )
   END_RUNG
   // the same network as SCL:
   IF "DB_SUB_1_ELEVADOR".Estados[13] AND "iSns_ElevAbajo" AND NOT Alarmas THEN
       "qCls_SoportRed" := FALSE;
   END_IF;
END_REGION

REGION Network 47: Retraigo lados
   RUNG wire#powerrail
      Contact( "DB_SUB_1_ELEVADOR".Estados[13] )
      Contact( "iSns_ElevAbajo" )
      I_Contact( Alarmas )
      S_Coil( "qOpn_Lados" )
   END_RUNG
   // the same network as SCL:
   IF "DB_SUB_1_ELEVADOR".Estados[13] AND "iSns_ElevAbajo" AND NOT Alarmas THEN "qOpn_Lados" := TRUE; END_IF;
END_REGION

REGION Network 48: Timer espera para abajar elevador
   "IEC_Timer_7_DB".TON(IN := "DB_SUB_1_ELEVADOR".Estados[13] AND "iSns_ElevAbajo" AND NOT Alarmas AND "qOpn_Lados",
                        PT := T#500MS);
   "B_TimAperturaLados" := "IEC_Timer_7_DB".Q;
END_REGION

REGION Network 49: Bajo elevador (normal)
   RUNG wire#powerrail
      Contact( "DB_SUB_1_ELEVADOR".Estados[14] )
      Contact( "B_TimAperturaLados" )
      I_Contact( Alarmas )
      Coil( "Bajo elevador" )
   END_RUNG
   // the same network as SCL:
   "Bajo elevador" := "DB_SUB_1_ELEVADOR".Estados[14] AND "B_TimAperturaLados" AND NOT Alarmas;
END_REGION
END_FUNCTION_BLOCK

FUNCTION_BLOCK "FB_SUB_1_CAMAS_ROLOS"   // FB102, LAD
{ S7_Optimized_Access := 'TRUE' }
VERSION : 0.1
BEGIN

REGION Network 2: --------------------------------------INSTANCIADO DE SUBSISTEMAS ---------------------------------------------------------
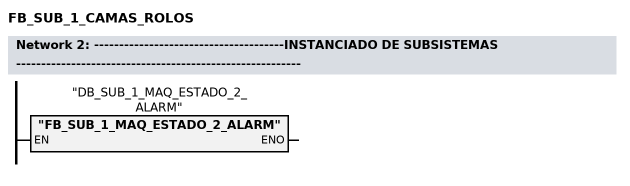
   RUNG wire#powerrail
      "DB_SUB_1_MAQ_ESTADO_2_ALARM"()
   END_RUNG
   // the same network as SCL:
   "DB_SUB_1_MAQ_ESTADO_2_ALARM"();   // "FB_SUB_1_MAQ_ESTADO_2_ALARM"
END_REGION

REGION Network 3: ------------------------------ ESTADOS DE LA MAQUINA - auto/manual -------------------------------------
END_REGION

REGION Network 9: --------------------------------------OTROS ---------------------------------------------------------
END_REGION

REGION Network 16: --------------------------------------MAQUINA DE ESTADOS ---------------------------------------------------------
END_REGION

REGION Network 29: --------------------------------------ACCIONAMIENTOS ---------------------------------------------------------
END_REGION
END_FUNCTION_BLOCK

FUNCTION_BLOCK "FB_SUB_1_MAQUINA_ESTADOS_3"   // FB103, LAD
{ S7_Optimized_Access := 'TRUE' }
VERSION : 0.1
BEGIN

REGION Network 1: --------------------------------------INSTANCIADO DE SUBSISTEMAS ---------------------------------------------------------
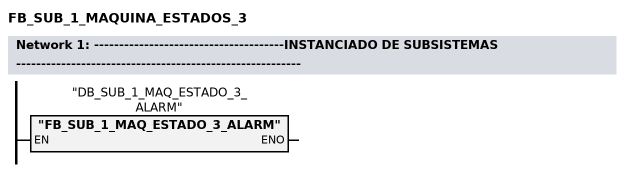
   RUNG wire#powerrail
      "DB_SUB_1_MAQ_ESTADO_3_ALARM"()
   END_RUNG
   // the same network as SCL:
   "DB_SUB_1_MAQ_ESTADO_3_ALARM"();   // "FB_SUB_1_MAQ_ESTADO_3_ALARM"
END_REGION

REGION Network 2: ------------------------------ ESTADOS DE LA MAQUINA - auto/manual -------------------------------------
END_REGION

REGION Network 8: --------------------------------------OTROS ---------------------------------------------------------
END_REGION

REGION Network 15: --------------------------------------MAQUINA DE ESTADOS ---------------------------------------------------------
END_REGION

REGION Network 28: --------------------------------------ACCIONAMIENTOS ---------------------------------------------------------
END_REGION
END_FUNCTION_BLOCK

FUNCTION_BLOCK "FB_SUB_1_MAQUINA_ESTADOS_4"   // FB104, LAD
{ S7_Optimized_Access := 'TRUE' }
VERSION : 0.1
BEGIN
END_FUNCTION_BLOCK

ORGANIZATION_BLOCK "Main"   // OB1, LAD, ProgramCycle
TITLE = "Main Program Sweep (Cycle)"
{ S7_Optimized_Access := 'TRUE' }
VERSION : 0.1
   VAR_INPUT
      Initial_Call : Bool;   // Initial call of this OB
      Remanence : Bool;   // =True, if remanent data are available
   END_VAR
   VAR_TEMP
      RetVal : Int;
   END_VAR
   VAR_TEMP   // added for the SCL form of the ladder/FBD networks
      _w1 : Bool;
   END_VAR
BEGIN

REGION Network 1: Instanciado subsistema "FB_SUB_0_GENERAL"
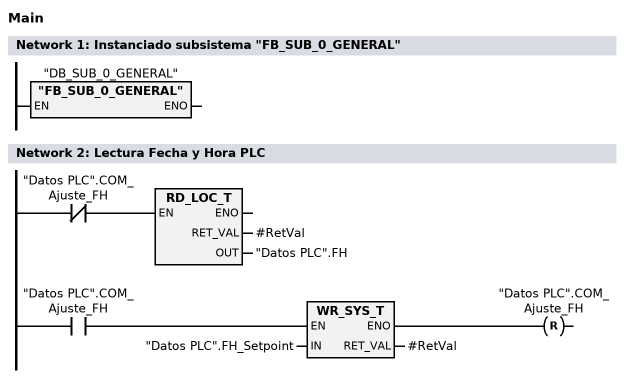
   RUNG wire#powerrail
      "DB_SUB_0_GENERAL"()
   END_RUNG
   // the same network as SCL:
   "DB_SUB_0_GENERAL"();   // "FB_SUB_0_GENERAL"
END_REGION

REGION Network 2: Lectura Fecha y Hora PLC
   // ENO of a box is taken as its EN; it also drops when the box reports an error
   IF NOT "Datos PLC".COM_Ajuste_FH THEN #RetVal := RD_LOC_T(OUT => "Datos PLC".FH); END_IF;
   #_w1 := "Datos PLC".COM_Ajuste_FH;
   IF #_w1 THEN
       #RetVal := WR_SYS_T(IN := "Datos PLC".FH_Setpoint);
       "Datos PLC".COM_Ajuste_FH := FALSE;
   END_IF;
END_REGION
END_ORGANIZATION_BLOCK

// folder: ENCLAVAMIENTOS

FUNCTION "FC_SUB_0_ENC_GENERAL" : Void   // FC700, LAD
{ S7_Optimized_Access := 'TRUE' }
VERSION : 0.1
BEGIN
END_FUNCTION

FUNCTION "FC_SUB_1_ENC_MAQ_ESTADOS_1" : Void   // FC701, LAD
{ S7_Optimized_Access := 'TRUE' }
VERSION : 0.1
BEGIN
END_FUNCTION

FUNCTION "FC_SUB_1_ENC_MAQ_ESTADOS_2" : Void   // FC702, LAD
{ S7_Optimized_Access := 'TRUE' }
VERSION : 0.1
BEGIN
END_FUNCTION

FUNCTION "FC_SUB_1_ENC_MAQ_ESTADOS_3" : Void   // FC703, LAD
{ S7_Optimized_Access := 'TRUE' }
VERSION : 0.1
BEGIN
END_FUNCTION

FUNCTION "FC_SUB_1_ENC_MAQ_ESTADOS_4" : Void   // FC704, LAD
{ S7_Optimized_Access := 'TRUE' }
VERSION : 0.1
BEGIN
END_FUNCTION

// folder: ESTANDAR

FUNCTION_BLOCK "Motor M&CM"   // FB2, LAD
TITLE = Motor Marcha & Contra-Marcha
{ S7_Optimized_Access := 'TRUE' }
VERSION : 0.1
   VAR_INPUT
      iOrdMar_Dir : Bool;
      iOrdMar_Rev : Bool;
      iConfMar_Dir : Bool;
      iConfMar_Rev : Bool;
      iGMT : Bool;
      iTConf_Warn : Time;
      iTConf_Fall : Time;
      iTRearranque : Time;
   END_VAR
   VAR_OUTPUT
      oMar_Dir : Bool;
      oMar_Rev : Bool;
      oWarning_CTC_Dir : Bool;
      oWarning_CTC_Rev : Bool;
      oFall_CTC_Dir : Bool;
      oFall_CTC_Rev : Bool;
      oFall_GMT : Bool;
   END_VAR
   VAR
      IEC_Timer_0_Instance : IEC_TIMER;
      IEC_Timer_0_Instance_1 : IEC_TIMER;
      IEC_Timer_0_Instance_2 : IEC_TIMER;
      IEC_Timer_0_Instance_3 : IEC_TIMER;
      IEC_Timer_0_Instance_4 : IEC_TIMER;
      MarDir_Aux : Bool;
      MarRev_Aux : Bool;
   END_VAR
   VAR_TEMP
      Fall_GMT_Aux : Bool;
      Fall_CTC_Dir_Aux : Bool;
      Fall_CTC_Rev_Aux : Bool;
      Habil_Mov : Bool;
   END_VAR
   VAR_TEMP   // added for the SCL form of the ladder/FBD networks
      _w1 : Bool;
   END_VAR
BEGIN

REGION Network 1: Falla Guardamotor
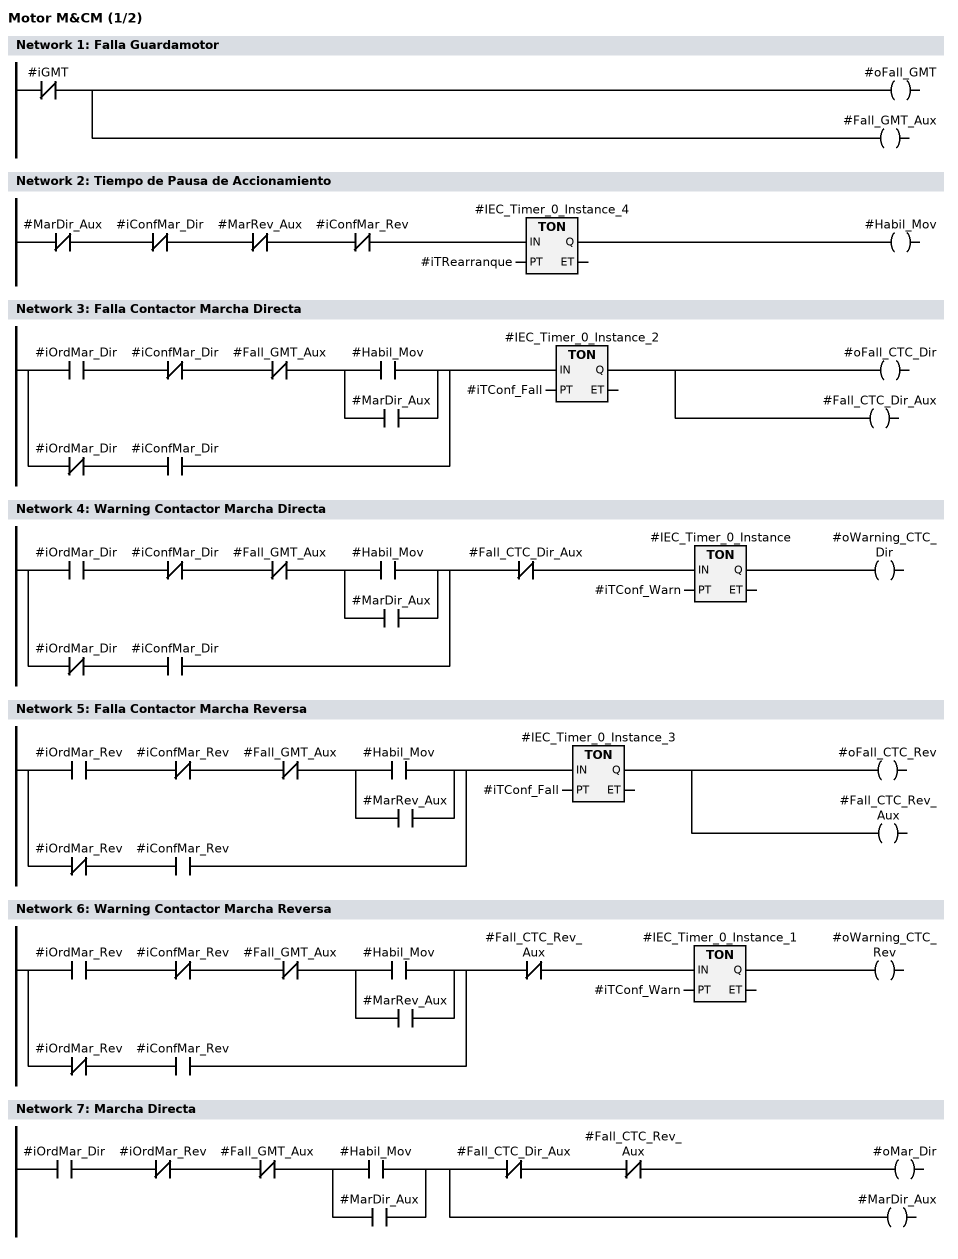
   RUNG wire#powerrail
      I_Contact( #iGMT )
      wire#w1
      Coil( #oFall_GMT )
   END_RUNG
   RUNG wire#w1
      Coil( #Fall_GMT_Aux )
   END_RUNG
   // the same network as SCL:
   #oFall_GMT := NOT #iGMT;
   #Fall_GMT_Aux := NOT #iGMT;
END_REGION

REGION Network 2: Tiempo de Pausa de Accionamiento
   #IEC_Timer_0_Instance_4.TON(IN := NOT #MarDir_Aux AND NOT #iConfMar_Dir AND NOT #MarRev_Aux AND NOT #iConfMar_Rev,
                           PT := #iTRearranque);
   #Habil_Mov := #IEC_Timer_0_Instance_4.Q;
END_REGION

REGION Network 3: Falla Contactor Marcha Directa
   #IEC_Timer_0_Instance_2.TON(IN := (#iOrdMar_Dir AND NOT #iConfMar_Dir AND NOT #Fall_GMT_Aux AND (#Habil_Mov OR #MarDir_Aux)) OR (NOT #iOrdMar_Dir AND #iConfMar_Dir),
                           PT := #iTConf_Fall);
   #oFall_CTC_Dir := #IEC_Timer_0_Instance_2.Q;
   #Fall_CTC_Dir_Aux := #IEC_Timer_0_Instance_2.Q;
END_REGION

REGION Network 4: Warning Contactor Marcha Directa
   #IEC_Timer_0_Instance.TON(IN := ((#iOrdMar_Dir AND NOT #iConfMar_Dir AND NOT #Fall_GMT_Aux AND (#Habil_Mov OR #MarDir_Aux)) OR (NOT #iOrdMar_Dir AND #iConfMar_Dir)) AND NOT #Fall_CTC_Dir_Aux,
                           PT := #iTConf_Warn);
   #oWarning_CTC_Dir := #IEC_Timer_0_Instance.Q;
END_REGION

REGION Network 5: Falla Contactor Marcha Reversa
   #IEC_Timer_0_Instance_3.TON(IN := (#iOrdMar_Rev AND NOT #iConfMar_Rev AND NOT #Fall_GMT_Aux AND (#Habil_Mov OR #MarRev_Aux)) OR (NOT #iOrdMar_Rev AND #iConfMar_Rev),
                           PT := #iTConf_Fall);
   #oFall_CTC_Rev := #IEC_Timer_0_Instance_3.Q;
   #Fall_CTC_Rev_Aux := #IEC_Timer_0_Instance_3.Q;
END_REGION

REGION Network 6: Warning Contactor Marcha Reversa
   #IEC_Timer_0_Instance_1.TON(IN := ((#iOrdMar_Rev AND NOT #iConfMar_Rev AND NOT #Fall_GMT_Aux AND (#Habil_Mov OR #MarRev_Aux)) OR (NOT #iOrdMar_Rev AND #iConfMar_Rev)) AND NOT #Fall_CTC_Rev_Aux,
                           PT := #iTConf_Warn);
   #oWarning_CTC_Rev := #IEC_Timer_0_Instance_1.Q;
END_REGION

REGION Network 7: Marcha Directa
   RUNG wire#powerrail
      Contact( #iOrdMar_Dir )
      I_Contact( #iOrdMar_Rev )
      I_Contact( #Fall_GMT_Aux )
      wire#w1
      Contact( #Habil_Mov )
      wire#w2
      I_Contact( #Fall_CTC_Dir_Aux )
      I_Contact( #Fall_CTC_Rev_Aux )
      Coil( #oMar_Dir )
   END_RUNG
   RUNG wire#w1
      Contact( #MarDir_Aux )
   END_RUNG wire#w2
   RUNG wire#w2
      Coil( #MarDir_Aux )
   END_RUNG
   // the same network as SCL:
   #_w1 := #iOrdMar_Dir AND NOT #iOrdMar_Rev AND NOT #Fall_GMT_Aux AND (#Habil_Mov OR #MarDir_Aux);
   #oMar_Dir := #_w1 AND NOT #Fall_CTC_Dir_Aux AND NOT #Fall_CTC_Rev_Aux;
   #MarDir_Aux := #_w1;
END_REGION

REGION Network 8: Marcha Reversa
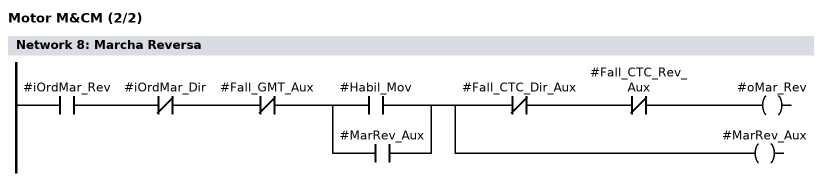
   RUNG wire#powerrail
      Contact( #iOrdMar_Rev )
      I_Contact( #iOrdMar_Dir )
      I_Contact( #Fall_GMT_Aux )
      wire#w1
      Contact( #Habil_Mov )
      wire#w2
      I_Contact( #Fall_CTC_Dir_Aux )
      I_Contact( #Fall_CTC_Rev_Aux )
      Coil( #oMar_Rev )
   END_RUNG
   RUNG wire#w1
      Contact( #MarRev_Aux )
   END_RUNG wire#w2
   RUNG wire#w2
      Coil( #MarRev_Aux )
   END_RUNG
   // the same network as SCL:
   #_w1 := #iOrdMar_Rev AND NOT #iOrdMar_Dir AND NOT #Fall_GMT_Aux AND (#Habil_Mov OR #MarRev_Aux);
   #oMar_Rev := #_w1 AND NOT #Fall_CTC_Dir_Aux AND NOT #Fall_CTC_Rev_Aux;
   #MarRev_Aux := #_w1;
END_REGION
END_FUNCTION_BLOCK

FUNCTION_BLOCK "FB_VAR_MOT"   // FB4, LAD
{ S7_Optimized_Access := 'FALSE' }
VERSION : 0.1
   VAR_INPUT
      "CMD Mar Dir" : Bool;   // Comando Marcha Directa
      "CMD Mar Rev" : Bool;   // Comando Marcha Reversa
      "HAB  Mar" : Bool;   // Habilita Marcha
      "SP Vel" : Real;   // Setpoint de Velocidad
      Reset : Bool;   // Comando resetear falla
      Fault : Bool;   // Indica variador en falla
      Ready : Bool;   // Indica variador Ready
      Ton_Freno : Time := T#400ms;
      Ton_Mar : Time := T#100ms;
      Tof_Freno : Time := T#100ms;
      Tof_Mar : Time := T#200ms;
   END_VAR
   VAR_OUTPUT
      Marcha : Bool;   // Orden de marcha a variador
      "Inv Giro" : Bool;   // Orden de invertir sentido de giro a variador
      "Reset Fault" : Bool;   // Reset Fault a variador
      Velocidad : Word;   // Referencia de Velocidad a variador
      Freno : Bool;   // Apertura de Freno
      Falla : Bool;   // Indica falla del variador
      Warning : Bool;   // Indica variador no Ready
   END_VAR
   VAR
      IEC_Timer_Freno : TON_TIME;
      IEC_Timer_Motor : TON_TIME;
      IEC_Timer_Reset : TOF_TIME;
      "_CMD Marcha Dir" : Bool;
      "_CMD Marcha Rev" : Bool;
      _CMD_AbrirFreno : Bool;
      IEC_Timer_0_Instance : TON_TIME;
      IEC_Timer_0_Instance_1 : TOF_TIME;
      IEC_Timer_0_Instance_2 : TOF_TIME;
      Ord_Marcha : Bool;
      Mem_Inv : Bool;
   END_VAR
   VAR_TEMP
      Vel_Real : Real;
      Vel_Int : Int;
      _Hab_Abrir_Freno : Bool;
      "Pre Marcha" : Bool;
      Aux : Bool;
      Freno_Aux : Bool;
   END_VAR
   VAR_TEMP   // added for the SCL form of the ladder/FBD networks
      _w1 : Bool;
      _w2 : Bool;
      _w3 : Bool;
   END_VAR
BEGIN

REGION Network 1: #Aux
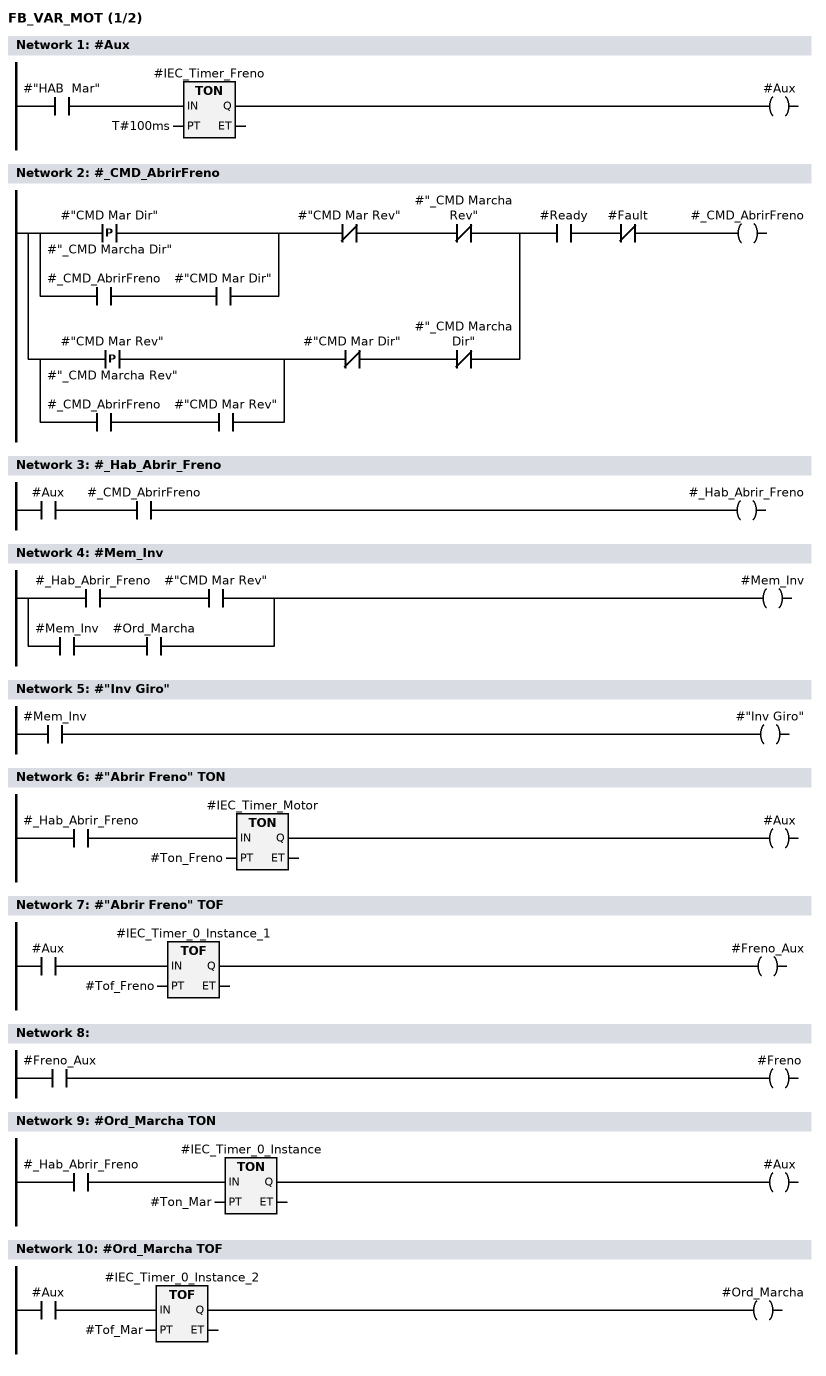
   #IEC_Timer_Freno(IN := #"HAB  Mar", PT := T#100ms);   // TON
   #Aux := #IEC_Timer_Freno.Q;
END_REGION

REGION Network 2: #_CMD_AbrirFreno
   RUNG wire#powerrail
      P_Contact(operand := #"CMD Mar Dir", bit := #"_CMD Marcha Dir")
      wire#w1
      I_Contact( #"CMD Mar Rev" )
      I_Contact( #"_CMD Marcha Rev" )
      wire#w2
      Contact( #Ready )
      I_Contact( #Fault )
      Coil( #_CMD_AbrirFreno )
   END_RUNG
   RUNG wire#powerrail
      Contact( #_CMD_AbrirFreno )
      Contact( #"CMD Mar Dir" )
   END_RUNG wire#w1
   RUNG wire#powerrail
      P_Contact(operand := #"CMD Mar Rev", bit := #"_CMD Marcha Rev")
      wire#w3
      I_Contact( #"CMD Mar Dir" )
      I_Contact( #"_CMD Marcha Dir" )
   END_RUNG wire#w2
   RUNG wire#powerrail
      Contact( #_CMD_AbrirFreno )
      Contact( #"CMD Mar Rev" )
   END_RUNG wire#w3
   // the same network as SCL:
   #_w1 := #"CMD Mar Dir" AND NOT #"_CMD Marcha Dir";   // rising edge of #"CMD Mar Dir"
   #"_CMD Marcha Dir" := #"CMD Mar Dir";
   #_w3 := (#_w1 OR (#_CMD_AbrirFreno AND #"CMD Mar Dir")) AND NOT #"CMD Mar Rev" AND NOT #"_CMD Marcha Rev";
   #_w2 := #"CMD Mar Rev" AND NOT #"_CMD Marcha Rev";   // rising edge of #"CMD Mar Rev"
   #"_CMD Marcha Rev" := #"CMD Mar Rev";
   #_CMD_AbrirFreno := (#_w3 OR ((#_w2 OR (#_CMD_AbrirFreno AND #"CMD Mar Rev")) AND NOT #"CMD Mar Dir" AND NOT #"_CMD Marcha Dir")) AND #Ready AND NOT #Fault;
END_REGION

REGION Network 3: #_Hab_Abrir_Freno
   RUNG wire#powerrail
      Contact( #Aux )
      Contact( #_CMD_AbrirFreno )
      Coil( #_Hab_Abrir_Freno )
   END_RUNG
   // the same network as SCL:
   #_Hab_Abrir_Freno := #Aux AND #_CMD_AbrirFreno;
END_REGION

REGION Network 4: #Mem_Inv
   RUNG wire#powerrail
      Contact( #_Hab_Abrir_Freno )
      Contact( #"CMD Mar Rev" )
      wire#w1
      Coil( #Mem_Inv )
   END_RUNG
   RUNG wire#powerrail
      Contact( #Mem_Inv )
      Contact( #Ord_Marcha )
   END_RUNG wire#w1
   // the same network as SCL:
   #Mem_Inv := (#_Hab_Abrir_Freno AND #"CMD Mar Rev") OR (#Mem_Inv AND #Ord_Marcha);
END_REGION

REGION Network 5: #"Inv Giro"
   RUNG wire#powerrail
      Contact( #Mem_Inv )
      Coil( #"Inv Giro" )
   END_RUNG
   // the same network as SCL:
   #"Inv Giro" := #Mem_Inv;
END_REGION

REGION Network 6: #"Abrir Freno" TON
   #IEC_Timer_Motor(IN := #_Hab_Abrir_Freno, PT := #Ton_Freno);   // TON
   #Aux := #IEC_Timer_Motor.Q;
END_REGION

REGION Network 7: #"Abrir Freno" TOF
   #IEC_Timer_0_Instance_1(IN := #Aux, PT := #Tof_Freno);   // TOF
   #Freno_Aux := #IEC_Timer_0_Instance_1.Q;
END_REGION

REGION Network 8
   RUNG wire#powerrail
      Contact( #Freno_Aux )
      Coil( #Freno )
   END_RUNG
   // the same network as SCL:
   #Freno := #Freno_Aux;
END_REGION

REGION Network 9: #Ord_Marcha TON
   #IEC_Timer_0_Instance(IN := #_Hab_Abrir_Freno, PT := #Ton_Mar);   // TON
   #Aux := #IEC_Timer_0_Instance.Q;
END_REGION

REGION Network 10: #Ord_Marcha TOF
   #IEC_Timer_0_Instance_2(IN := #Aux, PT := #Tof_Mar);   // TOF
   #Ord_Marcha := #IEC_Timer_0_Instance_2.Q;
END_REGION

REGION Network 11: #Marcha
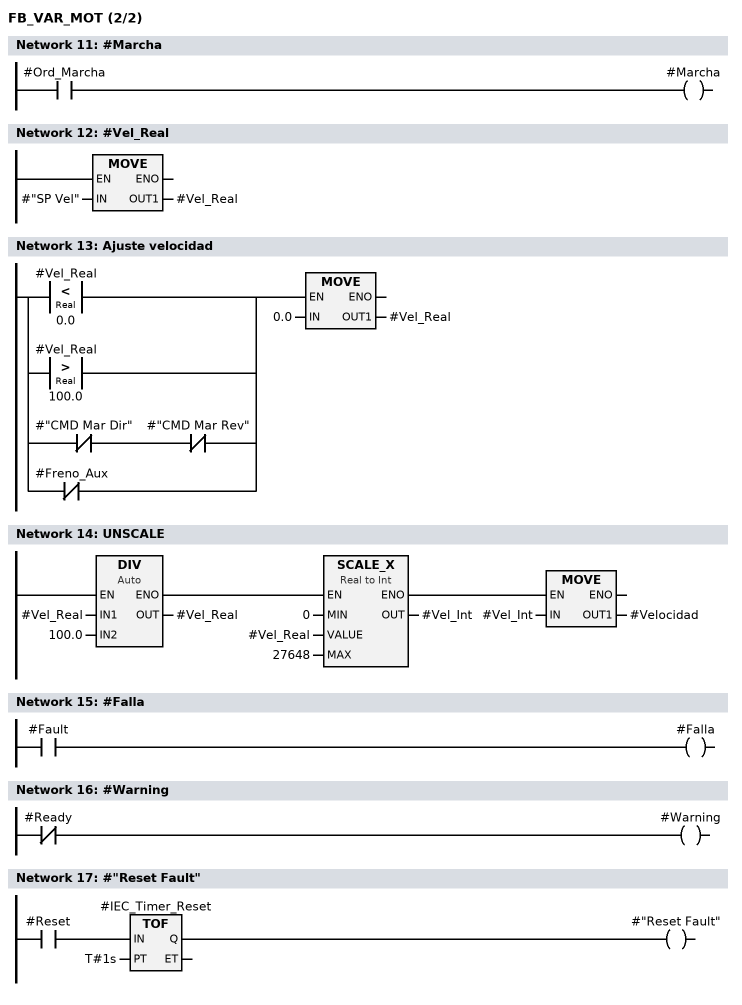
   RUNG wire#powerrail
      Contact( #Ord_Marcha )
      Coil( #Marcha )
   END_RUNG
   // the same network as SCL:
   #Marcha := #Ord_Marcha;
END_REGION

REGION Network 12: #Vel_Real
   RUNG wire#powerrail
      { S7_GenerateENO := "TRUE" } Move(in := #"SP Vel", out1 => #Vel_Real)
   END_RUNG
   // the same network as SCL:
   #Vel_Real := #"SP Vel";
END_REGION

REGION Network 13: Ajuste velocidad
   RUNG wire#powerrail
      { S7_Templates := "SrcType := Real" } LT_Contact(in1 := #Vel_Real, in2 := 0.0)
      wire#w1
      { S7_GenerateENO := "TRUE" } Move(in := 0.0, out1 => #Vel_Real)
   END_RUNG
   RUNG wire#powerrail
      { S7_Templates := "SrcType := Real" } GT_Contact(in1 := #Vel_Real, in2 := 100.0)
   END_RUNG wire#w1
   RUNG wire#powerrail
      I_Contact( #"CMD Mar Dir" )
      I_Contact( #"CMD Mar Rev" )
   END_RUNG wire#w1
   RUNG wire#powerrail
      I_Contact( #Freno_Aux )
   END_RUNG wire#w1
   // the same network as SCL:
   IF (#Vel_Real < 0.0) OR (#Vel_Real > 100.0) OR (NOT #"CMD Mar Dir" AND NOT #"CMD Mar Rev") OR NOT #Freno_Aux THEN
       #Vel_Real := 0.0;
   END_IF;
END_REGION

REGION Network 14: UNSCALE
   RUNG wire#powerrail
      Div(in1 := #Vel_Real, in2 := 100.0, out => #Vel_Real)
      { S7_Templates := "[SrcType := Real, DestType := Int]" } Scale(min := 0, value := #Vel_Real, max := 27648, out => #Vel_Int)
      { S7_GenerateENO := "TRUE" } Move(in := #Vel_Int, out1 => #Velocidad)
   END_RUNG
   // the same network as SCL:
   #Vel_Real := #Vel_Real / 100.0;
   #Vel_Int := SCALE_X(MIN := 0, VALUE := #Vel_Real, MAX := 27648);
   #Velocidad := #Vel_Int;
END_REGION

REGION Network 15: #Falla
   RUNG wire#powerrail
      Contact( #Fault )
      Coil( #Falla )
   END_RUNG
   // the same network as SCL:
   #Falla := #Fault;
END_REGION

REGION Network 16: #Warning
   RUNG wire#powerrail
      I_Contact( #Ready )
      Coil( #Warning )
   END_RUNG
   // the same network as SCL:
   #Warning := NOT #Ready;
END_REGION

REGION Network 17: #"Reset Fault"
   #IEC_Timer_Reset(IN := #Reset, PT := T#1s);   // TOF
   #"Reset Fault" := #IEC_Timer_Reset.Q;
END_REGION
END_FUNCTION_BLOCK

FUNCTION_BLOCK "Motor Simple"   // FB5, LAD
{ S7_Optimized_Access := 'TRUE' }
VERSION : 0.1
   VAR_INPUT
      iOrdMar : Bool;
      iConfMar : Bool;
      iGMT : Bool;
      iTConf_Warn : Time;
      iTConf_Fall : Time;
      iTRearranque : Time;
   END_VAR
   VAR_OUTPUT
      oMarcha : Bool;
      oWarning_CTC : Bool;
      oFall_CTC : Bool;
      oFall_GMT : Bool;
   END_VAR
   VAR
      IEC_Timer_0_Instance : IEC_TIMER;
      IEC_Timer_0_Instance_1 : IEC_TIMER;
      IEC_Timer_0_Instance_2 : IEC_TIMER;
      Mar_Aux : Bool;
   END_VAR
   VAR_TEMP
      Fall_GMT_Aux : Bool;
      Fall_CTC_Aux : Bool;
      Habil_Mov : Bool;
   END_VAR
BEGIN

REGION Network 1: Falla Guardamotor
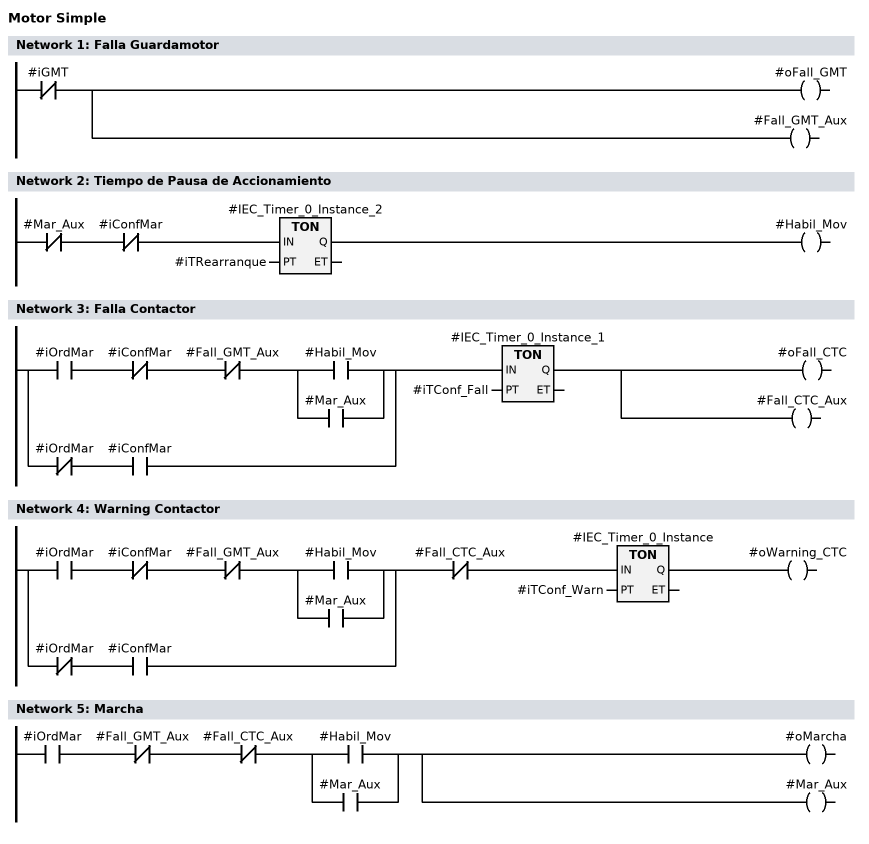
   RUNG wire#powerrail
      I_Contact( #iGMT )
      wire#w1
      Coil( #oFall_GMT )
   END_RUNG
   RUNG wire#w1
      Coil( #Fall_GMT_Aux )
   END_RUNG
   // the same network as SCL:
   #oFall_GMT := NOT #iGMT;
   #Fall_GMT_Aux := NOT #iGMT;
END_REGION

REGION Network 2: Tiempo de Pausa de Accionamiento
   #IEC_Timer_0_Instance_2.TON(IN := NOT #Mar_Aux AND NOT #iConfMar, PT := #iTRearranque);
   #Habil_Mov := #IEC_Timer_0_Instance_2.Q;
END_REGION

REGION Network 3: Falla Contactor
   #IEC_Timer_0_Instance_1.TON(IN := (#iOrdMar AND NOT #iConfMar AND NOT #Fall_GMT_Aux AND (#Habil_Mov OR #Mar_Aux)) OR (NOT #iOrdMar AND #iConfMar),
                           PT := #iTConf_Fall);
   #oFall_CTC := #IEC_Timer_0_Instance_1.Q;
   #Fall_CTC_Aux := #IEC_Timer_0_Instance_1.Q;
END_REGION

REGION Network 4: Warning Contactor
   #IEC_Timer_0_Instance.TON(IN := ((#iOrdMar AND NOT #iConfMar AND NOT #Fall_GMT_Aux AND (#Habil_Mov OR #Mar_Aux)) OR (NOT #iOrdMar AND #iConfMar)) AND NOT #Fall_CTC_Aux,
                           PT := #iTConf_Warn);
   #oWarning_CTC := #IEC_Timer_0_Instance.Q;
END_REGION

REGION Network 5: Marcha
   RUNG wire#powerrail
      Contact( #iOrdMar )
      I_Contact( #Fall_GMT_Aux )
      I_Contact( #Fall_CTC_Aux )
      wire#w1
      Contact( #Habil_Mov )
      wire#w2
      Coil( #oMarcha )
   END_RUNG
   RUNG wire#w1
      Contact( #Mar_Aux )
   END_RUNG wire#w2
   RUNG wire#w2
      Coil( #Mar_Aux )
   END_RUNG
   // the same network as SCL:
   #oMarcha := #iOrdMar AND NOT #Fall_GMT_Aux AND NOT #Fall_CTC_Aux AND (#Habil_Mov OR #Mar_Aux);
   #Mar_Aux := #oMarcha;
END_REGION
END_FUNCTION_BLOCK

FUNCTION_BLOCK "FB_VLV_2_POS"   // FB6, LAD
{ S7_Optimized_Access := 'FALSE' }
VERSION : 0.1
   VAR_INPUT
      Ir_Pos_1 : Bool;   // Comando Mover Cilindro a Posición 1, activar constantemente
      Ir_Pos_2 : Bool;   // Comando Mover Cilindro a Posición 2, activar constantemente
      Conf_Pos_1 : Bool;   // Confirmación Cilindro en Posición 1
      Conf_Pos_2 : Bool;   // Confirmación Cilindro en Posición 2
      T_Conf : Time := T#10s;   // Tiempo admisible para confirmación de posición
      T_ON : Time;   // Duración accionamiento salida [0 = constantemente]
   END_VAR
   VAR_OUTPUT
      Pos_1 : Bool;   // Orden Mover Cilindro a Posición 1
      Pos_2 : Bool;   // Orden Mover Cilindro a Posición 2
      ERROR : Int;   // 0 = Sin Error, 1 = Error Programación, 2 = Error Doble Confirmación, 3 = Error Confirmación Pos_1, 4 = Error Confirmación Pos_2, 5 = Sin Confirmaciones
   END_VAR
   VAR
      IEC_Timer_0_Instance : IEC_TIMER;
      IEC_Timer_0_Instance_1 : IEC_TIMER;
      IEC_Timer_0_Instance_2 : IEC_TIMER;
      IEC_Timer_0_Instance_3 : IEC_TIMER;
      IEC_Timer_0_Instance_4 : IEC_TIMER;
   END_VAR
   VAR_TEMP
      Aux_1 : Bool;   // Auxiliar 1
      Aux_2 : Bool;   // Auxiliar 2
      Aux_ERROR : Int;   // Auxiliar ERROR
   END_VAR
BEGIN

REGION Network 1: Auxiliar 1
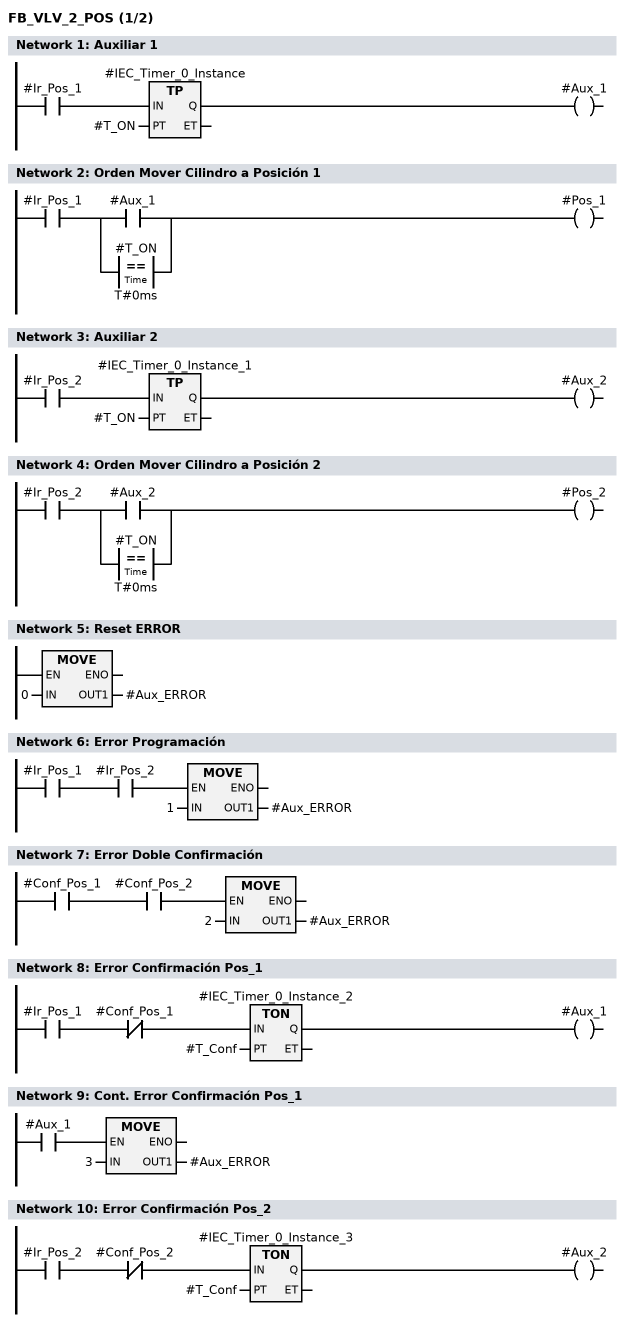
   #IEC_Timer_0_Instance.TP(IN := #Ir_Pos_1, PT := #T_ON);
   #Aux_1 := #IEC_Timer_0_Instance.Q;
END_REGION

REGION Network 2: Orden Mover Cilindro a Posición 1
   RUNG wire#powerrail
      Contact( #Ir_Pos_1 )
      wire#w1
      Contact( #Aux_1 )
      wire#w2
      Coil( #Pos_1 )
   END_RUNG
   RUNG wire#w1
      { S7_Templates := "SrcType := Time" } EQ_Contact(in1 := #T_ON, in2 := T#0ms)
   END_RUNG wire#w2
   // the same network as SCL:
   #Pos_1 := #Ir_Pos_1 AND (#Aux_1 OR (#T_ON = T#0ms));
END_REGION

REGION Network 3: Auxiliar 2
   #IEC_Timer_0_Instance_1.TP(IN := #Ir_Pos_2, PT := #T_ON);
   #Aux_2 := #IEC_Timer_0_Instance_1.Q;
END_REGION

REGION Network 4: Orden Mover Cilindro a Posición 2
   RUNG wire#powerrail
      Contact( #Ir_Pos_2 )
      wire#w1
      Contact( #Aux_2 )
      wire#w2
      Coil( #Pos_2 )
   END_RUNG
   RUNG wire#w1
      { S7_Templates := "SrcType := Time" } EQ_Contact(in1 := #T_ON, in2 := T#0ms)
   END_RUNG wire#w2
   // the same network as SCL:
   #Pos_2 := #Ir_Pos_2 AND (#Aux_2 OR (#T_ON = T#0ms));
END_REGION

REGION Network 5: Reset ERROR
   RUNG wire#powerrail
      { S7_GenerateENO := "TRUE" } Move(in := 0, out1 => #Aux_ERROR)
   END_RUNG
   // the same network as SCL:
   #Aux_ERROR := 0;
END_REGION

REGION Network 6: Error Programación
   RUNG wire#powerrail
      Contact( #Ir_Pos_1 )
      Contact( #Ir_Pos_2 )
      { S7_GenerateENO := "TRUE" } Move(in := 1, out1 => #Aux_ERROR)
   END_RUNG
   // the same network as SCL:
   IF #Ir_Pos_1 AND #Ir_Pos_2 THEN #Aux_ERROR := 1; END_IF;
END_REGION

REGION Network 7: Error Doble Confirmación
   RUNG wire#powerrail
      Contact( #Conf_Pos_1 )
      Contact( #Conf_Pos_2 )
      { S7_GenerateENO := "TRUE" } Move(in := 2, out1 => #Aux_ERROR)
   END_RUNG
   // the same network as SCL:
   IF #Conf_Pos_1 AND #Conf_Pos_2 THEN #Aux_ERROR := 2; END_IF;
END_REGION

REGION Network 8: Error Confirmación Pos_1
   #IEC_Timer_0_Instance_2.TON(IN := #Ir_Pos_1 AND NOT #Conf_Pos_1, PT := #T_Conf);
   #Aux_1 := #IEC_Timer_0_Instance_2.Q;
END_REGION

REGION Network 9: Cont. Error Confirmación Pos_1
   RUNG wire#powerrail
      Contact( #Aux_1 )
      { S7_GenerateENO := "TRUE" } Move(in := 3, out1 => #Aux_ERROR)
   END_RUNG
   // the same network as SCL:
   IF #Aux_1 THEN #Aux_ERROR := 3; END_IF;
END_REGION

REGION Network 10: Error Confirmación Pos_2
   #IEC_Timer_0_Instance_3.TON(IN := #Ir_Pos_2 AND NOT #Conf_Pos_2, PT := #T_Conf);
   #Aux_2 := #IEC_Timer_0_Instance_3.Q;
END_REGION

REGION Network 11: Cont. Error Confirmación Pos_2
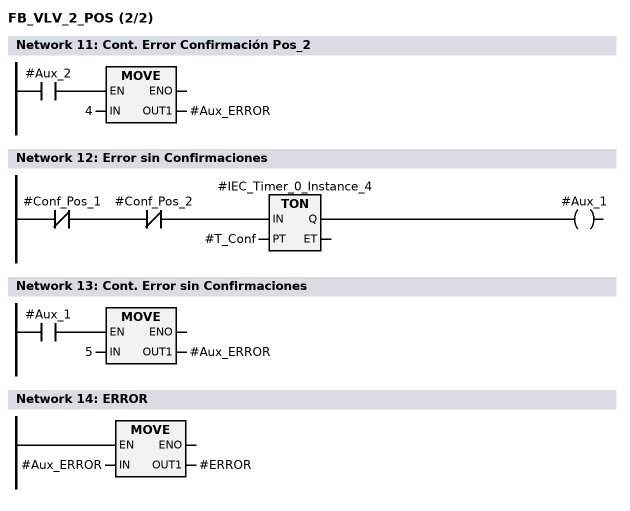
   RUNG wire#powerrail
      Contact( #Aux_2 )
      { S7_GenerateENO := "TRUE" } Move(in := 4, out1 => #Aux_ERROR)
   END_RUNG
   // the same network as SCL:
   IF #Aux_2 THEN #Aux_ERROR := 4; END_IF;
END_REGION

REGION Network 12: Error sin Confirmaciones
   #IEC_Timer_0_Instance_4.TON(IN := NOT #Conf_Pos_1 AND NOT #Conf_Pos_2, PT := #T_Conf);
   #Aux_1 := #IEC_Timer_0_Instance_4.Q;
END_REGION

REGION Network 13: Cont. Error sin Confirmaciones
   RUNG wire#powerrail
      Contact( #Aux_1 )
      { S7_GenerateENO := "TRUE" } Move(in := 5, out1 => #Aux_ERROR)
   END_RUNG
   // the same network as SCL:
   IF #Aux_1 THEN #Aux_ERROR := 5; END_IF;
END_REGION

REGION Network 14: ERROR
   RUNG wire#powerrail
      { S7_GenerateENO := "TRUE" } Move(in := #Aux_ERROR, out1 => #ERROR)
   END_RUNG
   // the same network as SCL:
   #ERROR := #Aux_ERROR;
END_REGION
END_FUNCTION_BLOCK

FUNCTION "MAQ_EST_32" : Void   // FC2, SCL
TITLE = Máquina de Estados 32
{ S7_Optimized_Access := 'TRUE' }
AUTHOR : FRD
FAMILY : MTA
NAME : MaqEst32
VERSION : 1.0
// KNOW_HOW_PROTECT  Máquina de estados de hasta 32 estados.
   VAR_INPUT
      Concatenadoras : DWord;   // Próximo estado de transición normal
      Prioritarias : DWord;   // Próximo estado de transición forzada
   END_VAR
   VAR_OUTPUT
      Error_Concatenadoras : Bool;   // Error en la programación de las Concatenadoras
      Error_Prioritarias : Bool;   // Error en la programación de las Prioritarias
   END_VAR
   VAR_IN_OUT
      Estado : DWord;   // Estado actual
   END_VAR
   VAR_TEMP
      Concat_Int : Int;   // Auxiliar INT para verificar las Concatenadoras
      Priorit_Int : Int;   // Auxiliar INT para verificar las Prioritarias
      Concat_Dword : DWord;   // Auxiliar DWORD para verificar las Concatenadoras
      Priorit_Dword : DWord;   // Auxiliar DWORD para verificar las Prioritarias
      Activar_Concat : Bool;   // Bit que indica Concatenadoras correctas
      Activar_Priorit : Bool;   // Bit que indica Prioritarias correctas
      Falla_Concat : Bool;   // Bit que indica falla en Concatenadoras
      Falla_Priorit : Bool;   // Bit que indica falla en Prioritarias
   END_VAR
BEGIN
   #Falla_Concat := 0;
   #Activar_Concat := 0;
   #Falla_Priorit := 0;
   #Activar_Priorit := 0; 
   #Error_Concatenadoras := 0;
   #Error_Prioritarias := 0;

   IF #Concatenadoras <> 0 THEN     //Evaluar Concatenadoras si son distintas de "0"

    #Concat_Int := ENCO(IN := #Concatenadoras );  //Convierte posición_DWORD en INT (0 a 31), lee el LSb

    #Concat_Dword := DECO(IN := INT_TO_UINT(#Concat_Int));//Convierte INT en posición_DWORD (1 a 32)

    IF #Concatenadoras = #Concat_Dword THEN  //Si son iguales, había sólo un bit en "1"

     #Activar_Concat := 1;    //Concatenadora correcta

    ELSE

     #Falla_Concat := 1;    //Falla en Concatenadora

    END_IF;

   END_IF;

   IF #Prioritarias <> 0 THEN     //Evaluar Prioritarias si son distintas de "0"

    #Priorit_Int := ENCO(IN := #Prioritarias);  //Convierte posición_DWORD en INT (0 a 31), lee el LSb

    #Priorit_Dword := DECO(IN := INT_TO_UINT(#Priorit_Int));//Convierte INT en posición_DWORD (1 a 32)

    IF #Prioritarias = #Priorit_Dword THEN  //Si son iguales, había sólo un bit en "1"

     #Activar_Priorit := 1;   //Prioritaria correcta

    ELSE

     #Falla_Priorit := 1;    //Falla en Prioritaria

    END_IF;

   END_IF;

   IF NOT(#Falla_Priorit OR #Falla_Concat) THEN  //Si no hay falla de Prioritaria ni de Concatenadora

    IF #Activar_Priorit THEN    //Si hay que asignar Prioritarias

     #Estado := #Prioritarias;

    ELSE

     IF #Activar_Concat THEN   //Si hay que asignar Concatenadoras

      #Estado := #Concatenadoras;

     END_IF;

    END_IF;

   ELSE

    IF #Falla_Concat THEN     //Si hay falla de Concatenadoras

     #Error_Concatenadoras := 1;    //Activar Error_Concatenadoras

    END_IF;

    IF #Falla_Priorit THEN    //Si hay falla de Prioritarias

     #Error_Prioritarias := 1;    //Activar Error_Prioritarias

    END_IF;

   END_IF;
END_FUNCTION

// folder: INCIDENTES

FUNCTION_BLOCK "FB_SUB_0_GENERAL_ALARM"   // FB1100, LAD
{ S7_Optimized_Access := 'TRUE' }
VERSION : 0.1
BEGIN
END_FUNCTION_BLOCK

FUNCTION_BLOCK "FB_SUB_1_MAQ_ESTADO_1_ALARM"   // FB1101, LAD
{ S7_Optimized_Access := 'TRUE' }
VERSION : 0.1
BEGIN
END_FUNCTION_BLOCK

FUNCTION_BLOCK "FB_SUB_1_MAQ_ESTADO_2_ALARM"   // FB1102, LAD
{ S7_Optimized_Access := 'TRUE' }
VERSION : 0.1
BEGIN
END_FUNCTION_BLOCK

FUNCTION_BLOCK "FB_SUB_1_MAQ_ESTADO_3_ALARM"   // FB1103, LAD
{ S7_Optimized_Access := 'TRUE' }
VERSION : 0.1
BEGIN
END_FUNCTION_BLOCK

FUNCTION_BLOCK "FB_SUB_1_MAQ_ESTADO_4_ALARM"   // FB1104, LAD
{ S7_Optimized_Access := 'TRUE' }
VERSION : 0.1
BEGIN

REGION Network 1: --------------------------------------INSTANCIADO DE SUBSISTEMAS ---------------------------------------------------------
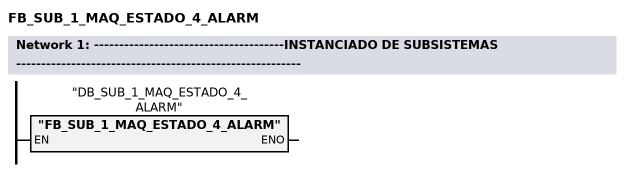
   RUNG wire#powerrail
      "DB_SUB_1_MAQ_ESTADO_4_ALARM"()
   END_RUNG
   // the same network as SCL:
   "DB_SUB_1_MAQ_ESTADO_4_ALARM"();   // "FB_SUB_1_MAQ_ESTADO_4_ALARM"
END_REGION

REGION Network 2: ------------------------------ ESTADOS DE LA MAQUINA - auto/manual -------------------------------------
END_REGION

REGION Network 8: --------------------------------------OTROS ---------------------------------------------------------
END_REGION

REGION Network 15: --------------------------------------MAQUINA DE ESTADOS ---------------------------------------------------------
END_REGION

REGION Network 28: --------------------------------------ACCIONAMIENTOS ---------------------------------------------------------
END_REGION
END_FUNCTION_BLOCK